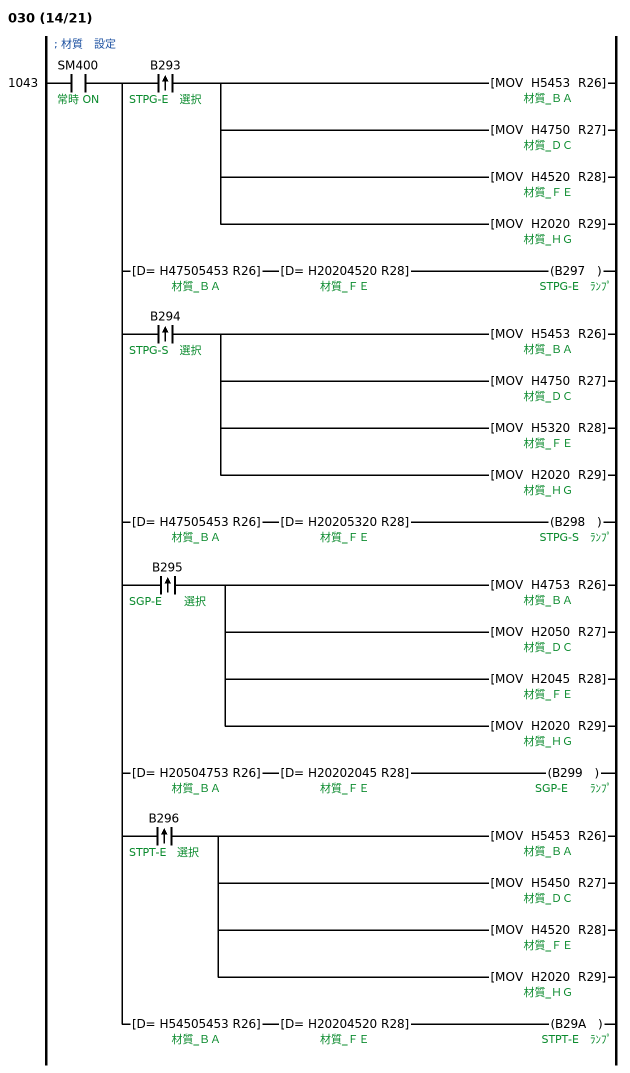
; 材質　設定
1043  LD      SM400  ; 常時 ON
      MPS
      ANDP    B293  ; STPG-E　選択
      MOV     H5453 R26  ; 材質_ＢＡ
      MOV     H4750 R27  ; 材質_ＤＣ
      MOV     H4520 R28  ; 材質_ＦＥ
      MOV     H2020 R29  ; 材質_ＨＧ
      MRD
      ANDD=   H47505453 R26  ; 材質_ＢＡ
      ANDD=   H20204520 R28  ; 材質_ＦＥ
      OUT     B297  ; STPG-E　ﾗﾝﾌﾟ
      MRD
      ANDP    B294  ; STPG-S　選択
      MOV     H5453 R26
      MOV     H4750 R27
      MOV     H5320 R28
      MOV     H2020 R29
      MRD
      ANDD=   H47505453 R26  ; 材質_ＢＡ
      ANDD=   H20205320 R28  ; 材質_ＦＥ
      OUT     B298  ; STPG-S　ﾗﾝﾌﾟ
      MRD
      ANDP    B295  ; SGP-E　　選択
      MOV     H4753 R26
      MOV     H2050 R27
      MOV     H2045 R28
      MOV     H2020 R29
      MRD
      ANDD=   H20504753 R26  ; 材質_ＢＡ
      ANDD=   H20202045 R28  ; 材質_ＦＥ
      OUT     B299  ; SGP-E　　ﾗﾝﾌﾟ
      MRD
      ANDP    B296  ; STPT-E　選択
      MOV     H5453 R26
      MOV     H5450 R27
      MOV     H4520 R28
      MOV     H2020 R29
      MPP
      ANDD=   H54505453 R26  ; 材質_ＢＡ
      ANDD=   H20204520 R28  ; 材質_ＦＥ
      OUT     B29A  ; STPT-E　ﾗﾝﾌﾟ
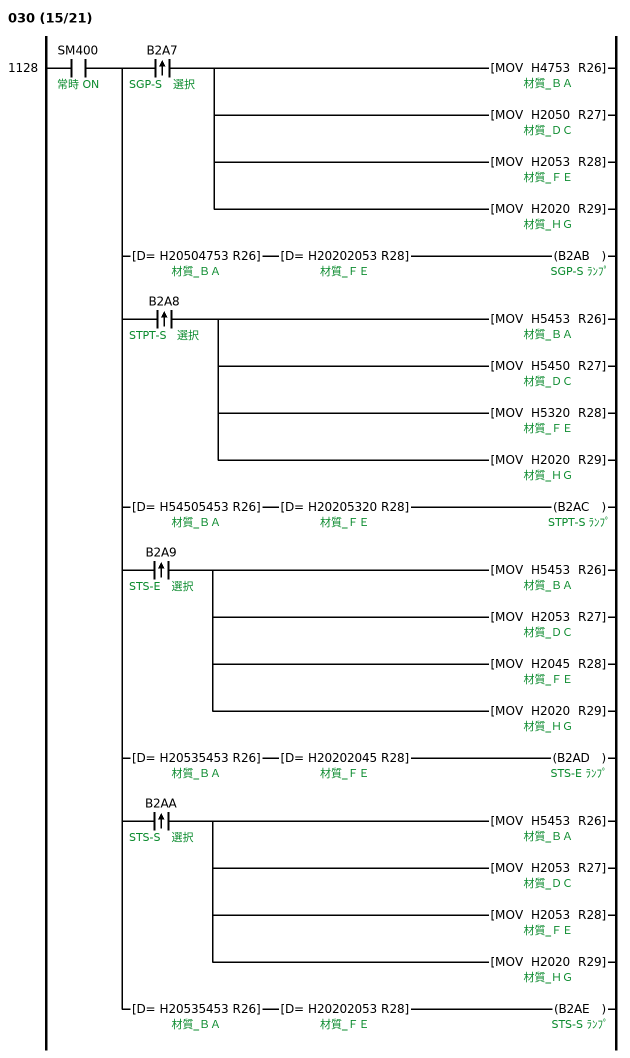
1128  LD      SM400  ; 常時 ON
      MPS
      ANDP    B2A7  ; SGP-S　選択
      MOV     H4753 R26
      MOV     H2050 R27
      MOV     H2053 R28
      MOV     H2020 R29
      MRD
      ANDD=   H20504753 R26  ; 材質_ＢＡ
      ANDD=   H20202053 R28  ; 材質_ＦＥ
      OUT     B2AB  ; SGP-S ﾗﾝﾌﾟ
      MRD
      ANDP    B2A8  ; STPT-S　選択
      MOV     H5453 R26
      MOV     H5450 R27
      MOV     H5320 R28
      MOV     H2020 R29
      MRD
      ANDD=   H54505453 R26  ; 材質_ＢＡ
      ANDD=   H20205320 R28  ; 材質_ＦＥ
      OUT     B2AC  ; STPT-S ﾗﾝﾌﾟ
      MRD
      ANDP    B2A9  ; STS-E　選択
      MOV     H5453 R26
      MOV     H2053 R27
      MOV     H2045 R28
      MOV     H2020 R29
      MRD
      ANDD=   H20535453 R26  ; 材質_ＢＡ
      ANDD=   H20202045 R28  ; 材質_ＦＥ
      OUT     B2AD  ; STS-E ﾗﾝﾌﾟ
      MRD
      ANDP    B2AA  ; STS-S　選択
      MOV     H5453 R26
      MOV     H2053 R27
      MOV     H2053 R28
      MOV     H2020 R29
      MPP
      ANDD=   H20535453 R26  ; 材質_ＢＡ
      ANDD=   H20202053 R28  ; 材質_ＦＥ
      OUT     B2AE  ; STS-S ﾗﾝﾌﾟ
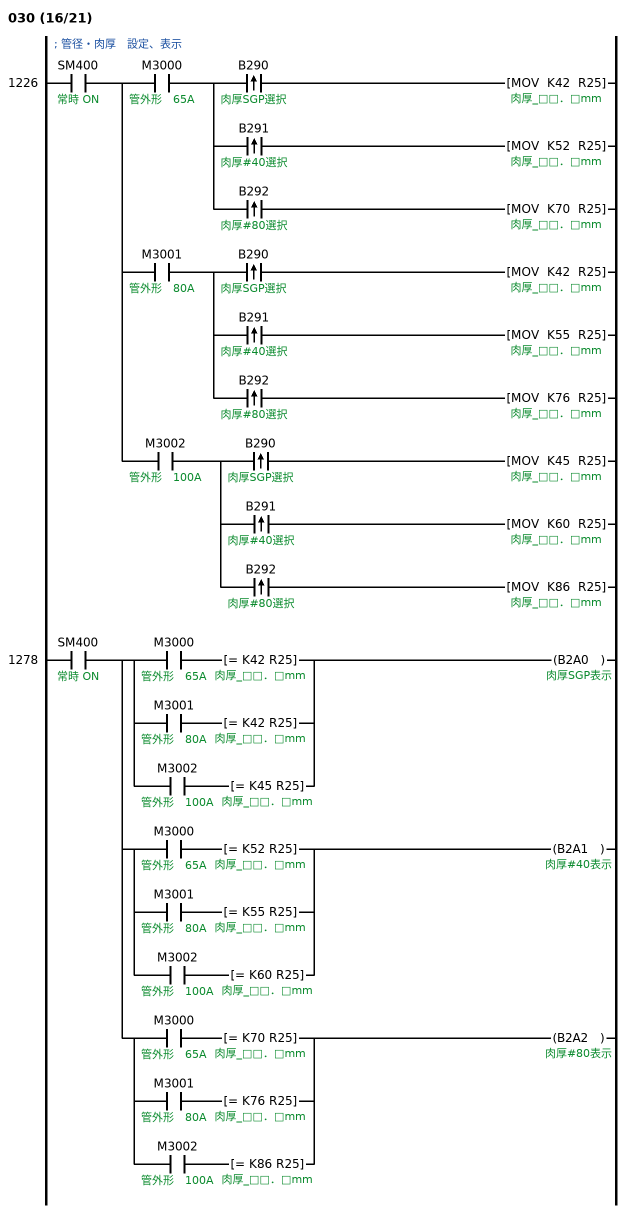
; 管径・肉厚　設定、表示
1226  LD      SM400  ; 常時 ON
      MPS
      AND     M3000  ; 管外形　65A
      MPS
      ANDP    B290  ; 肉厚SGP選択
      MOV     K42 R25  ; 肉厚_□□．□mm
      MRD
      ANDP    B291  ; 肉厚#40選択
      MOV     K52 R25
      MPP
      ANDP    B292  ; 肉厚#80選択
      MOV     K70 R25
      MRD
      AND     M3001  ; 管外形　80A
      MPS
      ANDP    B290  ; 肉厚SGP選択
      MOV     K42 R25
      MRD
      ANDP    B291  ; 肉厚#40選択
      MOV     K55 R25
      MPP
      ANDP    B292  ; 肉厚#80選択
      MOV     K76 R25
      MPP
      AND     M3002  ; 管外形　100A
      MPS
      ANDP    B290  ; 肉厚SGP選択
      MOV     K45 R25
      MRD
      ANDP    B291  ; 肉厚#40選択
      MOV     K60 R25
      MPP
      ANDP    B292  ; 肉厚#80選択
      MOV     K86 R25
1278  LD      SM400  ; 常時 ON
      MPS
      LD      M3000  ; 管外形　65A
      AND=    K42 R25  ; 肉厚_□□．□mm
      LD      M3001  ; 管外形　80A
      AND=    K42 R25  ; 肉厚_□□．□mm
      ORB
      LD      M3002  ; 管外形　100A
      AND=    K45 R25  ; 肉厚_□□．□mm
      ORB
      ANB
      OUT     B2A0  ; 肉厚SGP表示
      MRD
      LD      M3000  ; 管外形　65A
      AND=    K52 R25  ; 肉厚_□□．□mm
      LD      M3001  ; 管外形　80A
      AND=    K55 R25  ; 肉厚_□□．□mm
      ORB
      LD      M3002  ; 管外形　100A
      AND=    K60 R25  ; 肉厚_□□．□mm
      ORB
      ANB
      OUT     B2A1  ; 肉厚#40表示
      MPP
      LD      M3000  ; 管外形　65A
      AND=    K70 R25  ; 肉厚_□□．□mm
      LD      M3001  ; 管外形　80A
      AND=    K76 R25  ; 肉厚_□□．□mm
      ORB
      LD      M3002  ; 管外形　100A
      AND=    K86 R25  ; 肉厚_□□．□mm
      ORB
      ANB
      OUT     B2A2  ; 肉厚#80表示
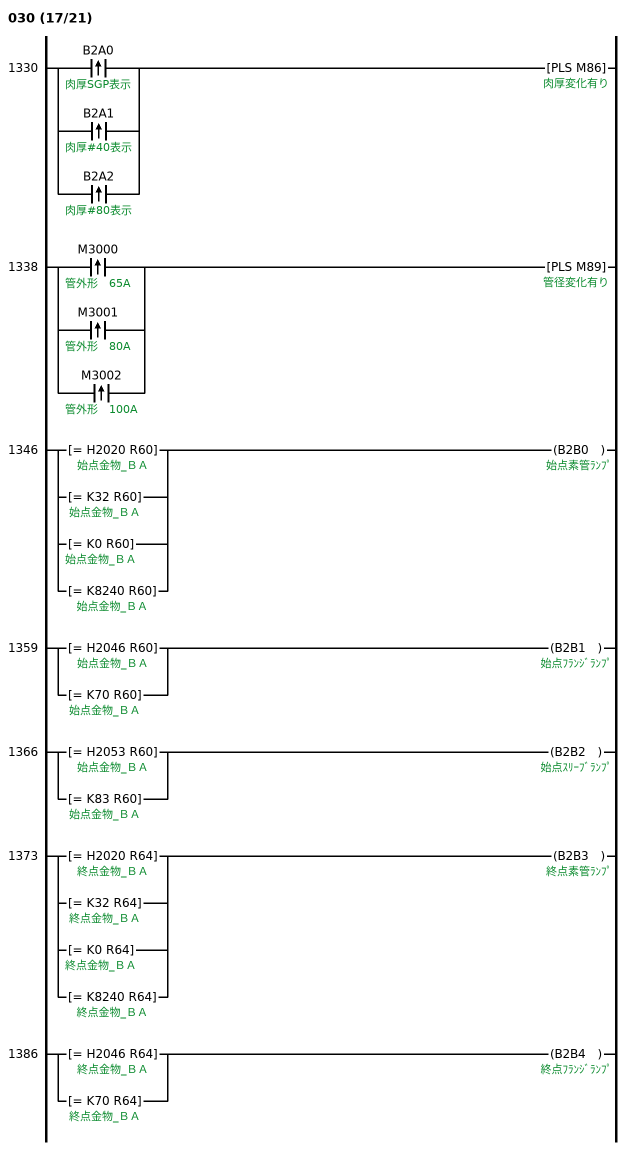
1330  LDP     B2A0  ; 肉厚SGP表示
      ORP     B2A1  ; 肉厚#40表示
      ORP     B2A2  ; 肉厚#80表示
      PLS     M86  ; 肉厚変化有り
1338  LDP     M3000  ; 管外形　65A
      ORP     M3001  ; 管外形　80A
      ORP     M3002  ; 管外形　100A
      PLS     M89  ; 管径変化有り
1346  LD=     H2020 R60  ; 始点金物_ＢＡ
      OR=     K32 R60  ; 始点金物_ＢＡ
      OR=     K0 R60  ; 始点金物_ＢＡ
      OR=     K8240 R60  ; 始点金物_ＢＡ
      OUT     B2B0  ; 始点素管ﾗﾝﾌﾟ
1359  LD=     H2046 R60  ; 始点金物_ＢＡ
      OR=     K70 R60  ; 始点金物_ＢＡ
      OUT     B2B1  ; 始点ﾌﾗﾝｼﾞﾗﾝﾌﾟ
1366  LD=     H2053 R60  ; 始点金物_ＢＡ
      OR=     K83 R60  ; 始点金物_ＢＡ
      OUT     B2B2  ; 始点ｽﾘｰﾌﾞﾗﾝﾌﾟ
1373  LD=     H2020 R64  ; 終点金物_ＢＡ
      OR=     K32 R64  ; 終点金物_ＢＡ
      OR=     K0 R64  ; 終点金物_ＢＡ
      OR=     K8240 R64  ; 終点金物_ＢＡ
      OUT     B2B3  ; 終点素管ﾗﾝﾌﾟ
1386  LD=     H2046 R64  ; 終点金物_ＢＡ
      OR=     K70 R64  ; 終点金物_ＢＡ
      OUT     B2B4  ; 終点ﾌﾗﾝｼﾞﾗﾝﾌﾟ
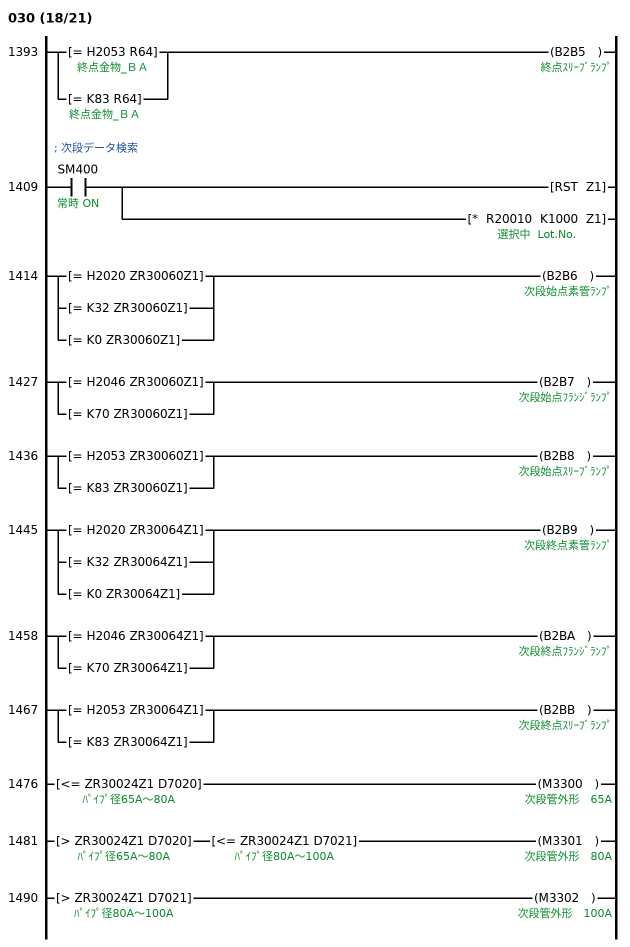
1393  LD=     H2053 R64  ; 終点金物_ＢＡ
      OR=     K83 R64  ; 終点金物_ＢＡ
      OUT     B2B5  ; 終点ｽﾘｰﾌﾞﾗﾝﾌﾟ
; 次段データ検索
1409  LD      SM400  ; 常時 ON
      RST     Z1
      *       R20010 K1000 Z1  ; 選択中  Lot.No.
1414  LD=     H2020 ZR30060Z1
      OR=     K32 ZR30060Z1
      OR=     K0 ZR30060Z1
      OUT     B2B6  ; 次段始点素管ﾗﾝﾌﾟ
1427  LD=     H2046 ZR30060Z1
      OR=     K70 ZR30060Z1
      OUT     B2B7  ; 次段始点ﾌﾗﾝｼﾞﾗﾝﾌﾟ
1436  LD=     H2053 ZR30060Z1
      OR=     K83 ZR30060Z1
      OUT     B2B8  ; 次段始点ｽﾘｰﾌﾞﾗﾝﾌﾟ
1445  LD=     H2020 ZR30064Z1
      OR=     K32 ZR30064Z1
      OR=     K0 ZR30064Z1
      OUT     B2B9  ; 次段終点素管ﾗﾝﾌﾟ
1458  LD=     H2046 ZR30064Z1
      OR=     K70 ZR30064Z1
      OUT     B2BA  ; 次段終点ﾌﾗﾝｼﾞﾗﾝﾌﾟ
1467  LD=     H2053 ZR30064Z1
      OR=     K83 ZR30064Z1
      OUT     B2BB  ; 次段終点ｽﾘｰﾌﾞﾗﾝﾌﾟ
1476  LD<=    ZR30024Z1 D7020  ; ﾊﾟｲﾌﾟ径65A～80A
      OUT     M3300  ; 次段管外形　65A
1481  LD>     ZR30024Z1 D7020  ; ﾊﾟｲﾌﾟ径65A～80A
      AND<=   ZR30024Z1 D7021  ; ﾊﾟｲﾌﾟ径80A～100A
      OUT     M3301  ; 次段管外形　80A
1490  LD>     ZR30024Z1 D7021  ; ﾊﾟｲﾌﾟ径80A～100A
      OUT     M3302  ; 次段管外形　100A
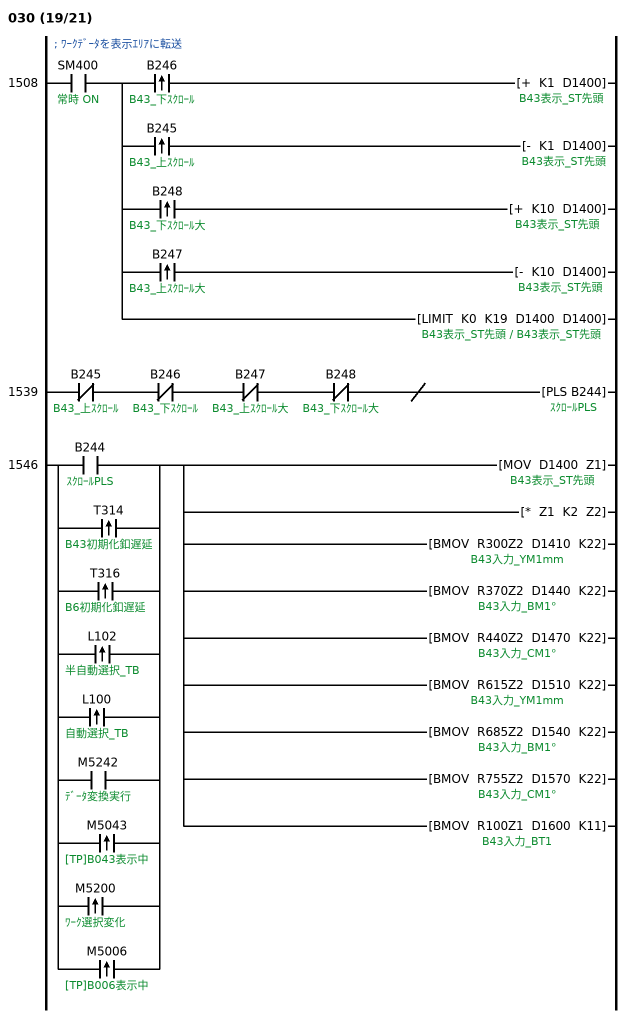
; ﾜｰｸﾃﾞｰﾀを表示ｴﾘｱに転送
1508  LD      SM400  ; 常時 ON
      MPS
      ANDP    B246  ; B43_下ｽｸﾛｰﾙ
      +       K1 D1400  ; B43表示_ST先頭
      MRD
      ANDP    B245  ; B43_上ｽｸﾛｰﾙ
      -       K1 D1400
      MRD
      ANDP    B248  ; B43_下ｽｸﾛｰﾙ大
      +       K10 D1400
      MRD
      ANDP    B247  ; B43_上ｽｸﾛｰﾙ大
      -       K10 D1400
      MPP
      LIMIT   K0 K19 D1400 D1400
1539  LDI     B245  ; B43_上ｽｸﾛｰﾙ
      ANI     B246  ; B43_下ｽｸﾛｰﾙ
      ANI     B247  ; B43_上ｽｸﾛｰﾙ大
      ANI     B248  ; B43_下ｽｸﾛｰﾙ大
      INV
      PLS     B244  ; ｽｸﾛｰﾙPLS
1546  LD      B244  ; ｽｸﾛｰﾙPLS
      ORP     T314  ; B43初期化釦遅延
      ORP     T316  ; B6初期化釦遅延
      ORP     L102  ; 半自動選択_TB
      ORP     L100  ; 自動選択_TB
      OR      M5242  ; ﾃﾞｰﾀ変換実行
      ORP     M5043  ; [TP]B043表示中
      ORP     M5200  ; ﾜｰｸ選択変化
      ORP     M5006  ; [TP]B006表示中
      MOV     D1400 Z1
      *       Z1 K2 Z2
      BMOV    R300Z2 D1410 K22  ; B43入力_YM1mm
      BMOV    R370Z2 D1440 K22  ; B43入力_BM1°
      BMOV    R440Z2 D1470 K22  ; B43入力_CM1°
      BMOV    R615Z2 D1510 K22  ; B43入力_YM1mm
      BMOV    R685Z2 D1540 K22  ; B43入力_BM1°
      BMOV    R755Z2 D1570 K22  ; B43入力_CM1°
      BMOV    R100Z1 D1600 K11  ; B43入力_BT1
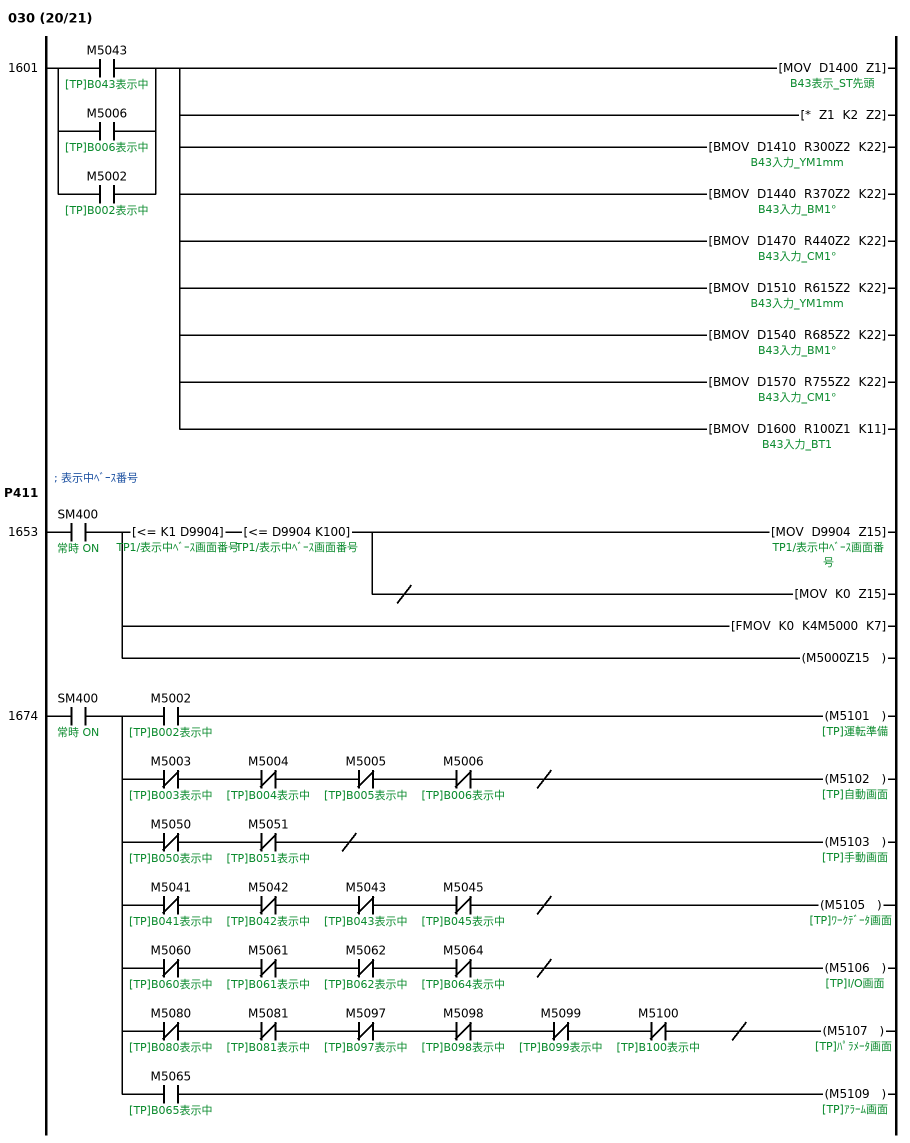
1601  LD      M5043  ; [TP]B043表示中
      OR      M5006  ; [TP]B006表示中
      OR      M5002  ; [TP]B002表示中
      MOV     D1400 Z1
      *       Z1 K2 Z2
      BMOV    D1410 R300Z2 K22
      BMOV    D1440 R370Z2 K22
      BMOV    D1470 R440Z2 K22
      BMOV    D1510 R615Z2 K22
      BMOV    D1540 R685Z2 K22
      BMOV    D1570 R755Z2 K22
      BMOV    D1600 R100Z1 K11
; 表示中ﾍﾞｰｽ番号
      P411
1653  LD      SM400  ; 常時 ON
      MPS
      AND<=   K1 D9904  ; TP1/表示中ﾍﾞｰｽ画面番号
      AND<=   D9904 K100  ; TP1/表示中ﾍﾞｰｽ画面番号
      MOV     D9904 Z15
      INV
      MOV     K0 Z15
      MPP
      FMOV    K0 K4M5000 K7  ; [TP]B00表示先頭
      OUT     M5000Z15
1674  LD      SM400  ; 常時 ON
      MPS
      AND     M5002  ; [TP]B002表示中
      OUT     M5101  ; [TP]運転準備
      MRD
      ANI     M5003  ; [TP]B003表示中
      ANI     M5004  ; [TP]B004表示中
      ANI     M5005  ; [TP]B005表示中
      ANI     M5006  ; [TP]B006表示中
      INV
      OUT     M5102  ; [TP]自動画面
      MRD
      ANI     M5050  ; [TP]B050表示中
      ANI     M5051  ; [TP]B051表示中
      INV
      OUT     M5103  ; [TP]手動画面
      MRD
      ANI     M5041  ; [TP]B041表示中
      ANI     M5042  ; [TP]B042表示中
      ANI     M5043  ; [TP]B043表示中
      ANI     M5045  ; [TP]B045表示中
      INV
      OUT     M5105  ; [TP]ﾜｰｸﾃﾞｰﾀ画面
      MRD
      ANI     M5060  ; [TP]B060表示中
      ANI     M5061  ; [TP]B061表示中
      ANI     M5062  ; [TP]B062表示中
      ANI     M5064  ; [TP]B064表示中
      INV
      OUT     M5106  ; [TP]I/O画面
      MRD
      ANI     M5080  ; [TP]B080表示中
      ANI     M5081  ; [TP]B081表示中
      ANI     M5097  ; [TP]B097表示中
      ANI     M5098  ; [TP]B098表示中
      ANI     M5099  ; [TP]B099表示中
      ANI     M5100  ; [TP]B100表示中
      INV
      OUT     M5107  ; [TP]ﾊﾟﾗﾒｰﾀ画面
      MPP
      AND     M5065  ; [TP]B065表示中
      OUT     M5109  ; [TP]ｱﾗｰﾑ画面
; 表示中ｳｨﾝﾄﾞｳ番号
      P412
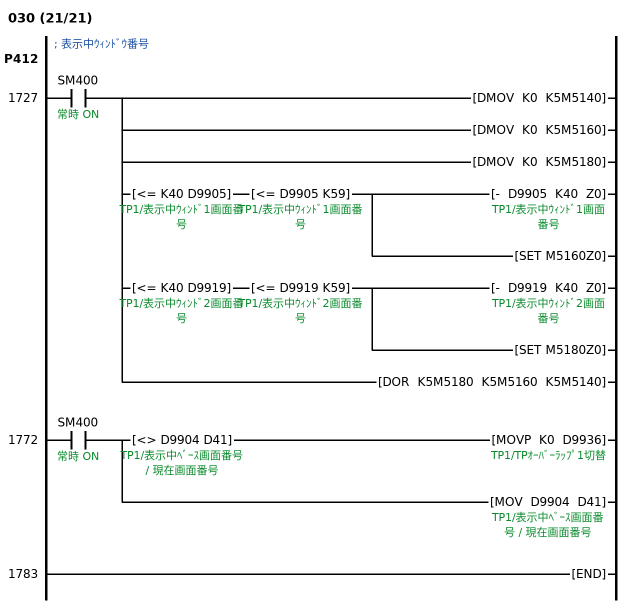
1727  LD      SM400  ; 常時 ON
      DMOV    K0 K5M5140  ; [TP]W40表示中
      DMOV    K0 K5M5160  ; WIN1_W40表示中
      DMOV    K0 K5M5180  ; WIN2_W40表示中
      MPS
      AND<=   K40 D9905  ; TP1/表示中ｳｨﾝﾄﾞ1画面番号
      AND<=   D9905 K59  ; TP1/表示中ｳｨﾝﾄﾞ1画面番号
      -       D9905 K40 Z0
      SET     M5160Z0
      MRD
      AND<=   K40 D9919  ; TP1/表示中ｳｨﾝﾄﾞ2画面番号
      AND<=   D9919 K59  ; TP1/表示中ｳｨﾝﾄﾞ2画面番号
      -       D9919 K40 Z0
      SET     M5180Z0
      MPP
      DOR     K5M5180 K5M5160 K5M5140
1772  LD      SM400  ; 常時 ON
      MPS
      AND<>   D9904 D41  ; TP1/表示中ﾍﾞｰｽ画面番号 / 現在画面番号
      MOVP    K0 D9936
      MPP
      MOV     D9904 D41
1783  END
END_PROGRAM

PROGRAM 031
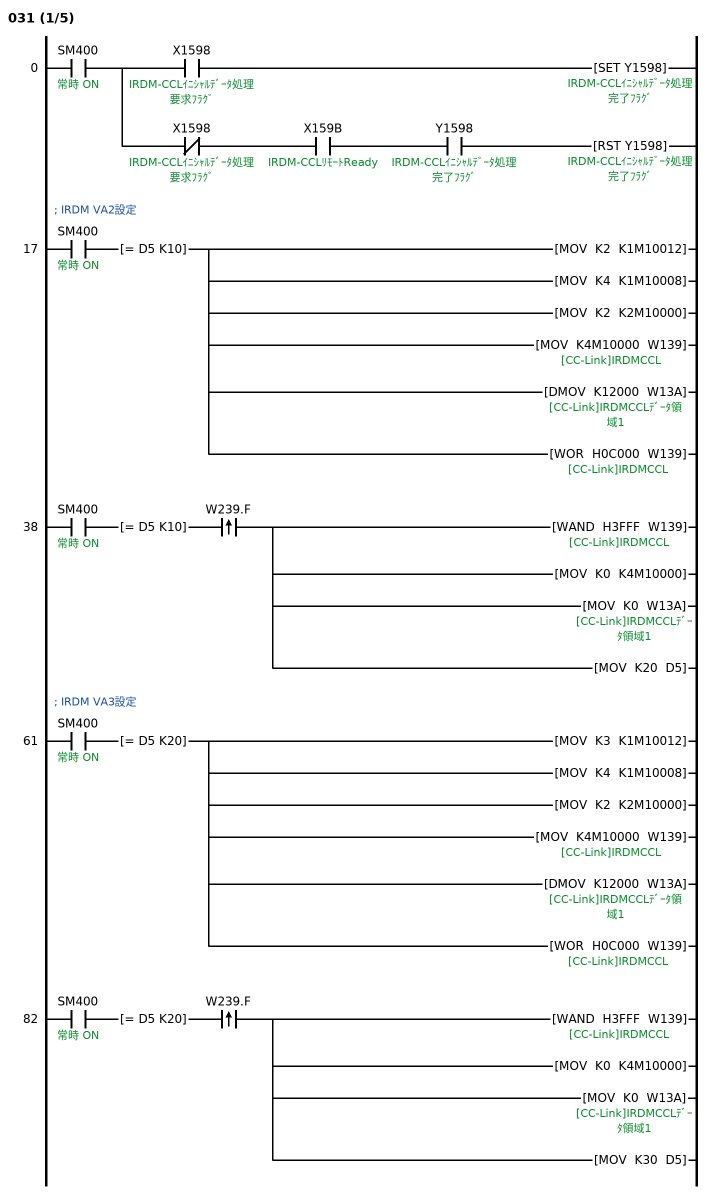
0     LD      SM400  ; 常時 ON
      MPS
      AND     X1598  ; IRDM-CCLｲﾆｼｬﾙﾃﾞｰﾀ処理要求ﾌﾗｸﾞ
      SET     Y1598  ; IRDM-CCLｲﾆｼｬﾙﾃﾞｰﾀ処理完了ﾌﾗｸﾞ
      MPP
      ANI     X1598  ; IRDM-CCLｲﾆｼｬﾙﾃﾞｰﾀ処理要求ﾌﾗｸﾞ
      AND     X159B  ; IRDM-CCLﾘﾓｰﾄReady
      AND     Y1598  ; IRDM-CCLｲﾆｼｬﾙﾃﾞｰﾀ処理完了ﾌﾗｸﾞ
      RST     Y1598  ; IRDM-CCLｲﾆｼｬﾙﾃﾞｰﾀ処理完了ﾌﾗｸﾞ
; IRDM VA2設定
17    LD      SM400  ; 常時 ON
      AND=    D5 K10
      MOV     K2 K1M10012  ; [IRDM仮変数]ﾁｬﾝﾈﾙ番号
      MOV     K4 K1M10008  ; [IRDM仮変数]ｸﾞﾙｰﾌﾟ番号
      MOV     K2 K2M10000  ; [IRDM仮変数]ｲﾝﾃﾞｯｸｽ番号
      MOV     K4M10000 W139  ; [CC-Link]IRDMCCL
      DMOV    K12000 W13A  ; [CC-Link]IRDMCCLﾃﾞｰﾀ領域1
      WOR     H0C000 W139
38    LD      SM400  ; 常時 ON
      AND=    D5 K10
      ANDP    W239.F
      WAND    H3FFF W139
      MOV     K0 K4M10000
      MOV     K0 W13A
      MOV     K20 D5
; IRDM VA3設定
61    LD      SM400  ; 常時 ON
      AND=    D5 K20
      MOV     K3 K1M10012
      MOV     K4 K1M10008
      MOV     K2 K2M10000
      MOV     K4M10000 W139
      DMOV    K12000 W13A
      WOR     H0C000 W139
82    LD      SM400  ; 常時 ON
      AND=    D5 K20
      ANDP    W239.F
      WAND    H3FFF W139
      MOV     K0 K4M10000
      MOV     K0 W13A
      MOV     K30 D5
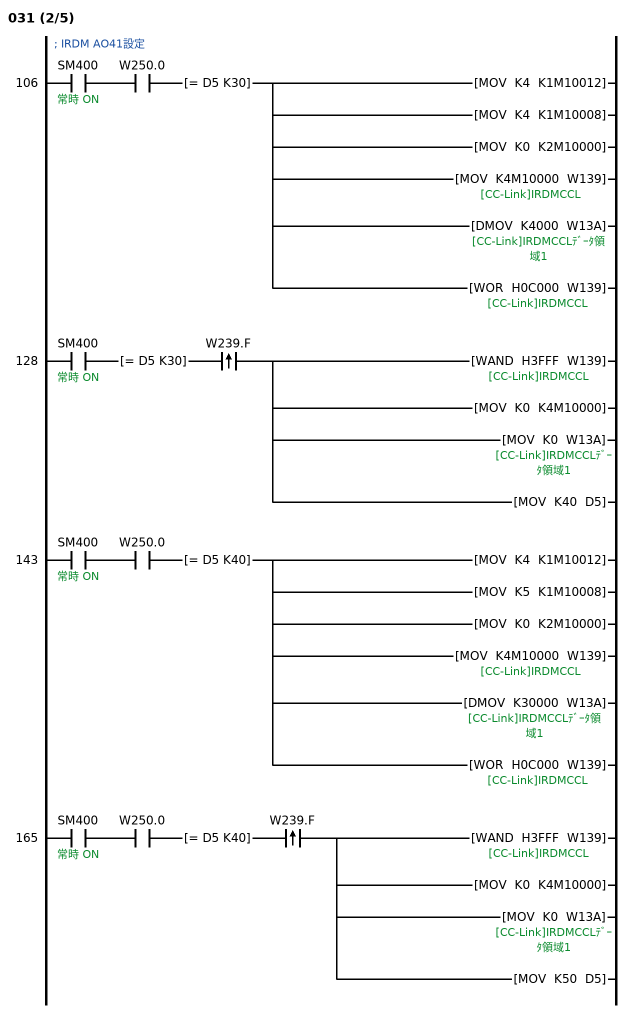
; IRDM AO41設定
106   LD      SM400  ; 常時 ON
      AND     W250.0
      AND=    D5 K30
      MOV     K4 K1M10012
      MOV     K4 K1M10008
      MOV     K0 K2M10000
      MOV     K4M10000 W139
      DMOV    K4000 W13A
      WOR     H0C000 W139
128   LD      SM400  ; 常時 ON
      AND=    D5 K30
      ANDP    W239.F
      WAND    H3FFF W139
      MOV     K0 K4M10000
      MOV     K0 W13A
      MOV     K40 D5
143   LD      SM400  ; 常時 ON
      AND     W250.0
      AND=    D5 K40
      MOV     K4 K1M10012
      MOV     K5 K1M10008
      MOV     K0 K2M10000
      MOV     K4M10000 W139
      DMOV    K30000 W13A
      WOR     H0C000 W139
165   LD      SM400  ; 常時 ON
      AND     W250.0
      AND=    D5 K40
      ANDP    W239.F
      WAND    H3FFF W139
      MOV     K0 K4M10000
      MOV     K0 W13A
      MOV     K50 D5
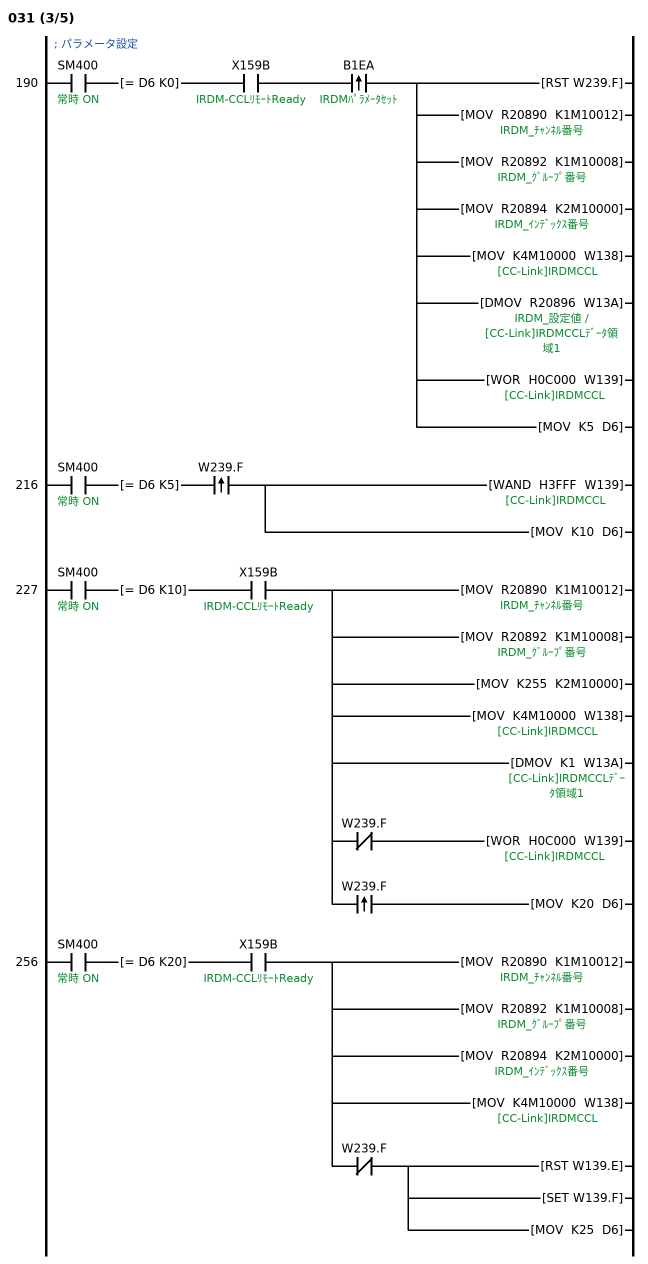
; パラメータ設定
190   LD      SM400  ; 常時 ON
      AND=    D6 K0
      AND     X159B  ; IRDM-CCLﾘﾓｰﾄReady
      ANDP    B1EA  ; IRDMﾊﾟﾗﾒｰﾀｾｯﾄ
      RST     W239.F
      MOV     R20890 K1M10012  ; IRDM_ﾁｬﾝﾈﾙ番号
      MOV     R20892 K1M10008  ; IRDM_ｸﾞﾙｰﾌﾟ番号
      MOV     R20894 K2M10000  ; IRDM_ｲﾝﾃﾞｯｸｽ番号
      MOV     K4M10000 W138  ; [CC-Link]IRDMCCL
      DMOV    R20896 W13A  ; IRDM_設定値
      WOR     H0C000 W139
      MOV     K5 D6
216   LD      SM400  ; 常時 ON
      AND=    D6 K5
      ANDP    W239.F
      WAND    H3FFF W139
      MOV     K10 D6
227   LD      SM400  ; 常時 ON
      AND=    D6 K10
      AND     X159B  ; IRDM-CCLﾘﾓｰﾄReady
      MOV     R20890 K1M10012
      MOV     R20892 K1M10008
      MOV     K255 K2M10000
      MOV     K4M10000 W138
      DMOV    K1 W13A
      MPS
      ANI     W239.F
      WOR     H0C000 W139
      MPP
      ANDP    W239.F
      MOV     K20 D6
256   LD      SM400  ; 常時 ON
      AND=    D6 K20
      AND     X159B  ; IRDM-CCLﾘﾓｰﾄReady
      MOV     R20890 K1M10012
      MOV     R20892 K1M10008
      MOV     R20894 K2M10000
      MOV     K4M10000 W138
      ANI     W239.F
      RST     W139.E
      SET     W139.F
      MOV     K25 D6
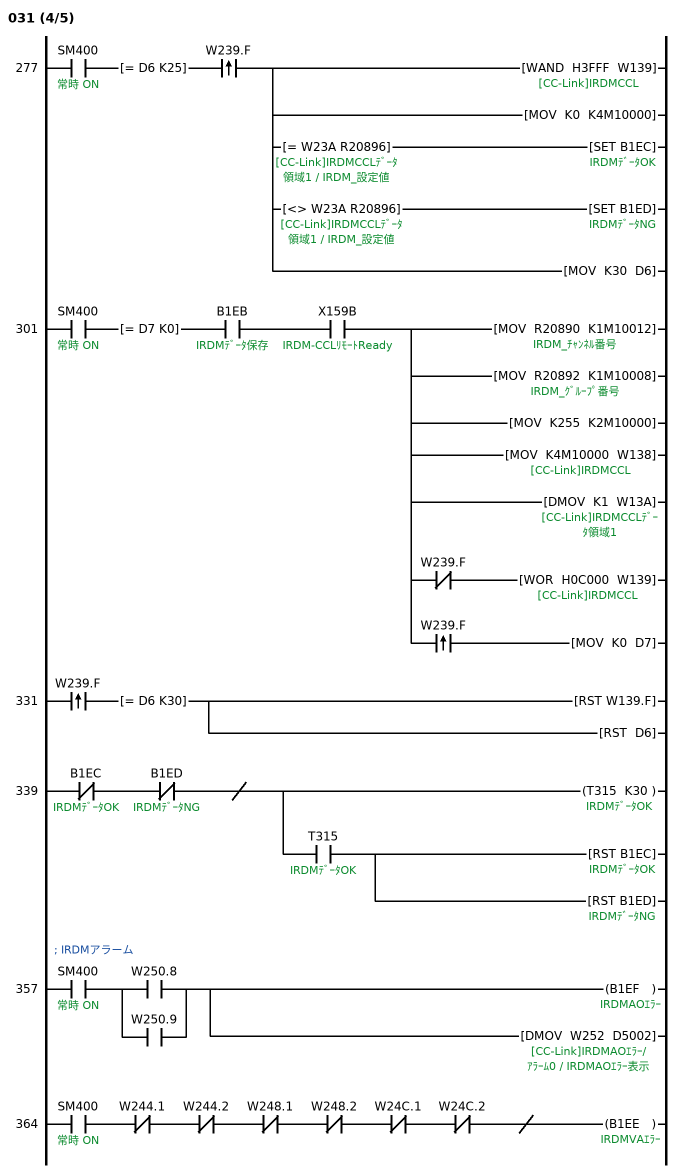
277   LD      SM400  ; 常時 ON
      AND=    D6 K25
      ANDP    W239.F
      WAND    H3FFF W139
      MOV     K0 K4M10000
      MPS
      AND=    W23A R20896  ; [CC-Link]IRDMCCLﾃﾞｰﾀ領域1 / IRDM_設定値
      SET     B1EC  ; IRDMﾃﾞｰﾀOK
      MRD
      AND<>   W23A R20896  ; [CC-Link]IRDMCCLﾃﾞｰﾀ領域1 / IRDM_設定値
      SET     B1ED  ; IRDMﾃﾞｰﾀNG
      MPP
      MOV     K30 D6
301   LD      SM400  ; 常時 ON
      AND=    D7 K0
      AND     B1EB  ; IRDMﾃﾞｰﾀ保存
      AND     X159B  ; IRDM-CCLﾘﾓｰﾄReady
      MOV     R20890 K1M10012
      MOV     R20892 K1M10008
      MOV     K255 K2M10000
      MOV     K4M10000 W138
      DMOV    K1 W13A
      MPS
      ANI     W239.F
      WOR     H0C000 W139
      MPP
      ANDP    W239.F
      MOV     K0 D7
331   LDP     W239.F
      AND=    D6 K30
      RST     W139.F
      RST     D6
339   LDI     B1EC  ; IRDMﾃﾞｰﾀOK
      ANI     B1ED  ; IRDMﾃﾞｰﾀNG
      INV
      OUT     T315 K30  ; IRDMﾃﾞｰﾀOK
      AND     T315  ; IRDMﾃﾞｰﾀOK
      RST     B1EC  ; IRDMﾃﾞｰﾀOK
      RST     B1ED  ; IRDMﾃﾞｰﾀNG
; IRDMアラーム
357   LD      SM400  ; 常時 ON
      LD      W250.8
      OR      W250.9
      ANB
      OUT     B1EF  ; IRDMAOｴﾗｰ
      DMOV    W252 D5002  ; [CC-Link]IRDMAOｴﾗｰ/ｱﾗｰﾑ0 / IRDMAOｴﾗｰ表示
364   LD      SM400  ; 常時 ON
      ANI     W244.1
      ANI     W244.2
      ANI     W248.1
      ANI     W248.2
      ANI     W24C.1
      ANI     W24C.2
      INV
      OUT     B1EE  ; IRDMVAｴﾗｰ
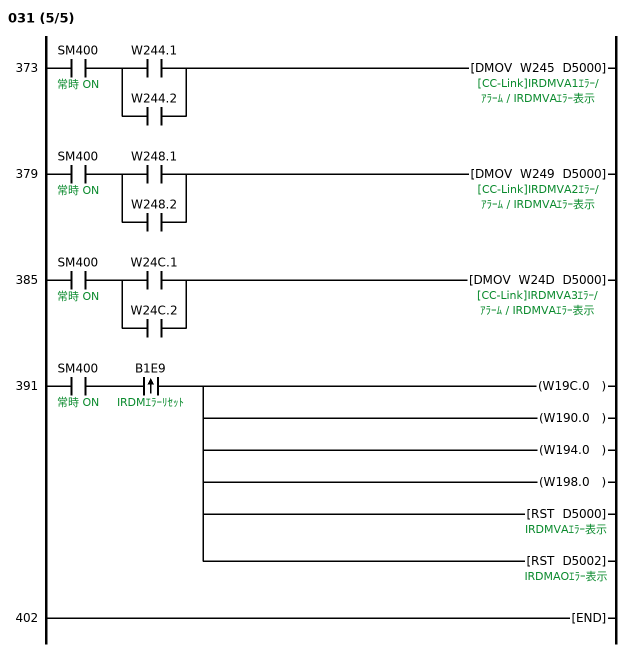
373   LD      SM400  ; 常時 ON
      LD      W244.1
      OR      W244.2
      ANB
      DMOV    W245 D5000  ; [CC-Link]IRDMVA1ｴﾗｰ/ｱﾗｰﾑ / IRDMVAｴﾗｰ表示
379   LD      SM400  ; 常時 ON
      LD      W248.1
      OR      W248.2
      ANB
      DMOV    W249 D5000  ; [CC-Link]IRDMVA2ｴﾗｰ/ｱﾗｰﾑ
385   LD      SM400  ; 常時 ON
      LD      W24C.1
      OR      W24C.2
      ANB
      DMOV    W24D D5000  ; [CC-Link]IRDMVA3ｴﾗｰ/ｱﾗｰﾑ
391   LD      SM400  ; 常時 ON
      ANDP    B1E9  ; IRDMｴﾗｰﾘｾｯﾄ
      OUT     W19C.0
      OUT     W190.0
      OUT     W194.0
      OUT     W198.0
      RST     D5000  ; IRDMVAｴﾗｰ表示
      RST     D5002  ; IRDMAOｴﾗｰ表示
402   END
END_PROGRAM

PROGRAM 016
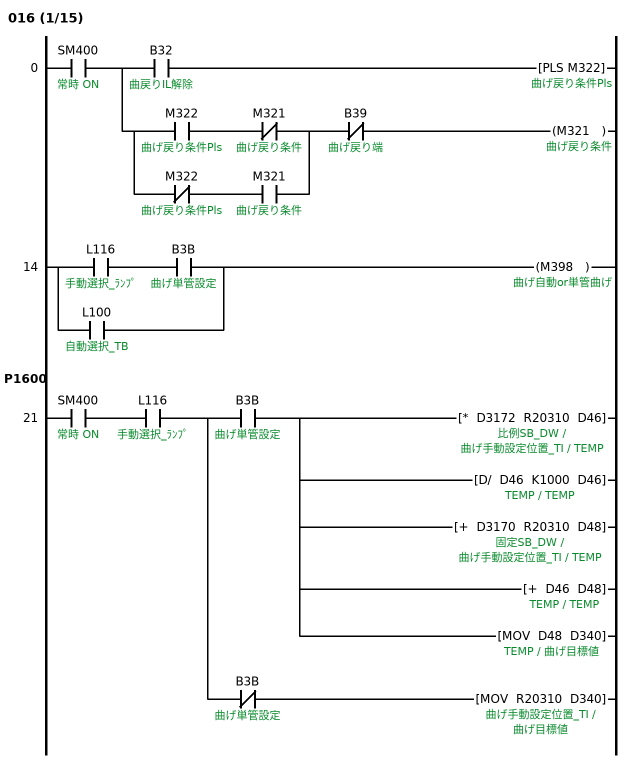
0     LD      SM400  ; 常時 ON
      MPS
      AND     B32  ; 曲戻りIL解除
      PLS     M322  ; 曲げ戻り条件Pls
      MPP
      LD      M322  ; 曲げ戻り条件Pls
      ANI     M321  ; 曲げ戻り条件
      LDI     M322  ; 曲げ戻り条件Pls
      AND     M321  ; 曲げ戻り条件
      ORB
      ANB
      ANI     B39  ; 曲げ戻り端
      OUT     M321  ; 曲げ戻り条件
14    LD      L116  ; 手動選択_ﾗﾝﾌﾟ
      AND     B3B  ; 曲げ単管設定
      OR      L100  ; 自動選択_TB
      OUT     M398  ; 曲げ自動or単管曲げ
; 
      P1600
21    LD      SM400  ; 常時 ON
      AND     L116  ; 手動選択_ﾗﾝﾌﾟ
      MPS
      AND     B3B  ; 曲げ単管設定
      *       D3172 R20310 D46  ; 比例SB_DW / 曲げ手動設定位置_TI / TEMP
      D/      D46 K1000 D46
      +       D3170 R20310 D48  ; 固定SB_DW / TEMP
      +       D46 D48
      MOV     D48 D340  ; 曲げ目標値
      MPP
      ANI     B3B  ; 曲げ単管設定
      MOV     R20310 D340
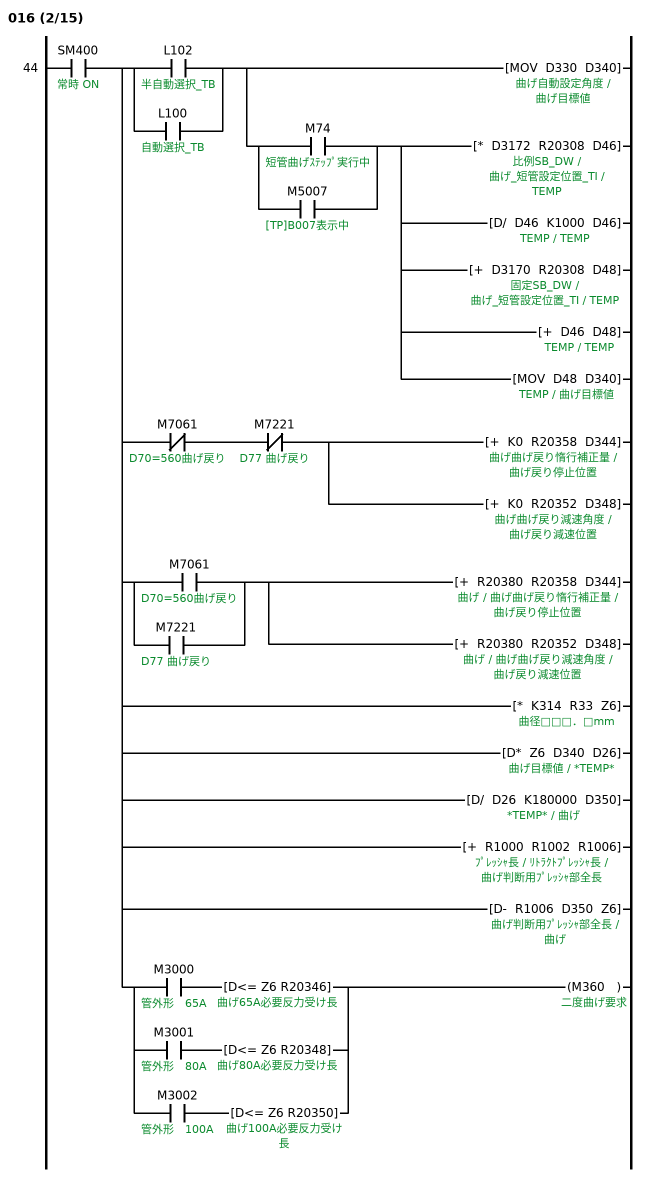
44    LD      SM400  ; 常時 ON
      MPS
      LD      L102  ; 半自動選択_TB
      OR      L100  ; 自動選択_TB
      ANB
      MOV     D330 D340  ; 曲げ自動設定角度
      LD      M74  ; 短管曲げｽﾃｯﾌﾟ実行中
      OR      M5007  ; [TP]B007表示中
      ANB
      *       D3172 R20308 D46  ; 曲げ_短管設定位置_TI
      D/      D46 K1000 D46
      +       D3170 R20308 D48
      +       D46 D48
      MOV     D48 D340
      MRD
      ANI     M7061  ; D70=560曲げ戻り
      ANI     M7221  ; D77 曲げ戻り
      +       K0 R20358 D344  ; 曲げ曲げ戻り惰行補正量 / 曲げ戻り停止位置
      +       K0 R20352 D348  ; 曲げ曲げ戻り減速角度 / 曲げ戻り減速位置
      MRD
      LD      M7061  ; D70=560曲げ戻り
      OR      M7221  ; D77 曲げ戻り
      ANB
      +       R20380 R20358 D344  ; 曲げ
      +       R20380 R20352 D348
      MPP
      *       K314 R33 Z6  ; 曲径□□□．□mm
      D*      Z6 D340 D26  ; *TEMP*
      D/      D26 K180000 D350  ; 曲げ
      +       R1000 R1002 R1006  ; ﾌﾟﾚｯｼｬ長 / ﾘﾄﾗｸﾄﾌﾟﾚｯｼｬ長 / 曲げ判断用ﾌﾟﾚｯｼｬ部全長
      D-      R1006 D350 Z6
      LD      M3000  ; 管外形　65A
      ANDD<=  Z6 R20346  ; 曲げ65A必要反力受け長
      LD      M3001  ; 管外形　80A
      ANDD<=  Z6 R20348  ; 曲げ80A必要反力受け長
      ORB
      LD      M3002  ; 管外形　100A
      ANDD<=  Z6 R20350  ; 曲げ100A必要反力受け長
      ORB
      ANB
      OUT     M360  ; 二度曲げ要求
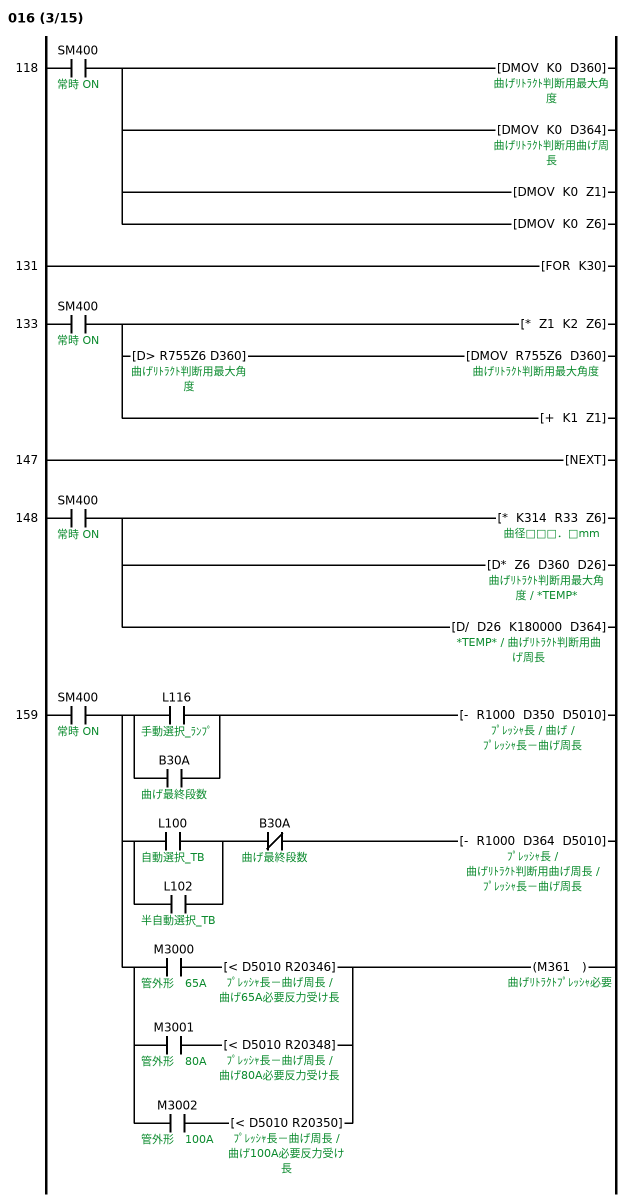
118   LD      SM400  ; 常時 ON
      DMOV    K0 D360  ; 曲げﾘﾄﾗｸﾄ判断用最大角度
      DMOV    K0 D364  ; 曲げﾘﾄﾗｸﾄ判断用曲げ周長
      DMOV    K0 Z1
      DMOV    K0 Z6
131   FOR     K30
133   LD      SM400  ; 常時 ON
      *       Z1 K2 Z6
      MPS
      ANDD>   R755Z6 D360  ; 曲げﾘﾄﾗｸﾄ判断用最大角度
      DMOV    R755Z6 D360
      MPP
      +       K1 Z1
147   NEXT
148   LD      SM400  ; 常時 ON
      *       K314 R33 Z6
      D*      Z6 D360 D26
      D/      D26 K180000 D364
159   LD      SM400  ; 常時 ON
      MPS
      LD      L116  ; 手動選択_ﾗﾝﾌﾟ
      OR      B30A  ; 曲げ最終段数
      ANB
      -       R1000 D350 D5010  ; ﾌﾟﾚｯｼｬ長－曲げ周長
      MRD
      LD      L100  ; 自動選択_TB
      OR      L102  ; 半自動選択_TB
      ANB
      ANI     B30A  ; 曲げ最終段数
      -       R1000 D364 D5010
      MPP
      LD      M3000  ; 管外形　65A
      AND<    D5010 R20346  ; ﾌﾟﾚｯｼｬ長－曲げ周長 / 曲げ65A必要反力受け長
      LD      M3001  ; 管外形　80A
      AND<    D5010 R20348  ; ﾌﾟﾚｯｼｬ長－曲げ周長 / 曲げ80A必要反力受け長
      ORB
      LD      M3002  ; 管外形　100A
      AND<    D5010 R20350  ; ﾌﾟﾚｯｼｬ長－曲げ周長 / 曲げ100A必要反力受け長
      ORB
      ANB
      OUT     M361  ; 曲げﾘﾄﾗｸﾄﾌﾟﾚｯｼｬ必要
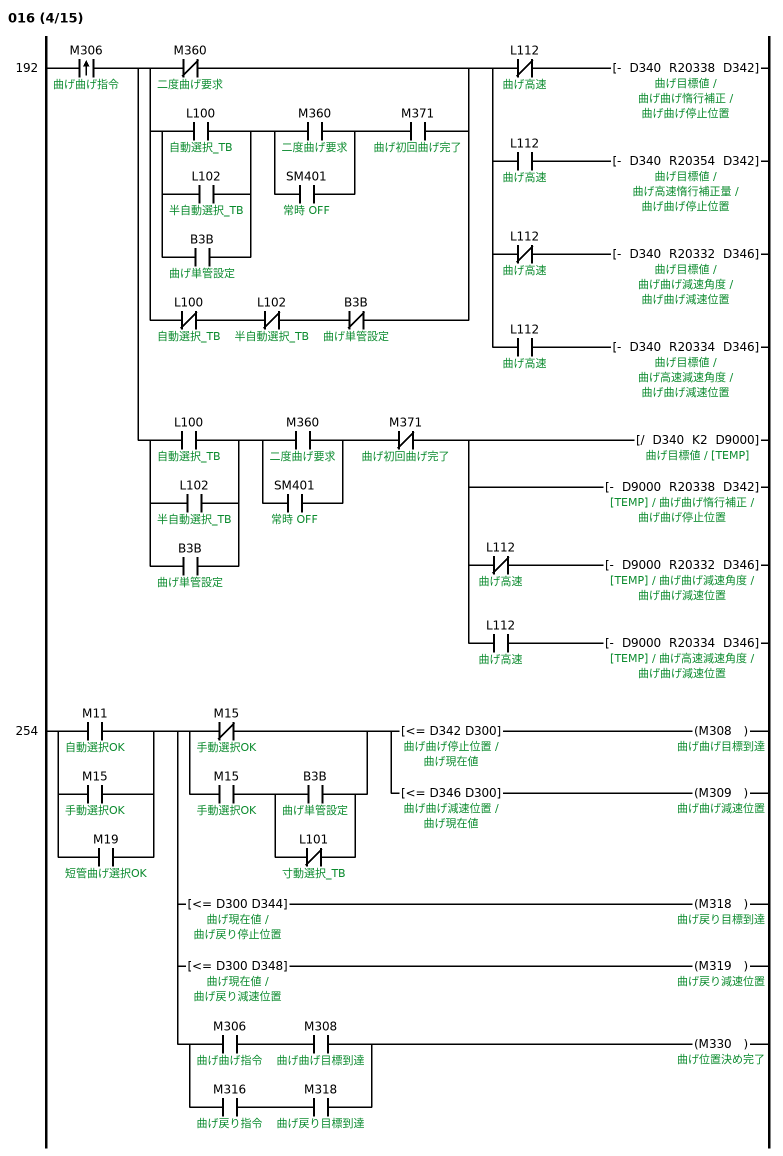
192   LDP     M306  ; 曲げ曲げ指令
      MPS
      LDI     M360  ; 二度曲げ要求
      LD      L100  ; 自動選択_TB
      OR      L102  ; 半自動選択_TB
      OR      B3B  ; 曲げ単管設定
      LD      M360  ; 二度曲げ要求
      OR      SM401  ; 常時 OFF
      ANB
      AND     M371  ; 曲げ初回曲げ完了
      ORB
      LDI     L100  ; 自動選択_TB
      ANI     L102  ; 半自動選択_TB
      ANI     B3B  ; 曲げ単管設定
      ORB
      ANB
      MPS
      ANI     L112  ; 曲げ高速
      -       D340 R20338 D342  ; 曲げ曲げ惰行補正 / 曲げ曲げ停止位置
      MRD
      AND     L112  ; 曲げ高速
      -       D340 R20354 D342  ; 曲げ高速惰行補正量
      MRD
      ANI     L112  ; 曲げ高速
      -       D340 R20332 D346  ; 曲げ曲げ減速角度 / 曲げ曲げ減速位置
      MPP
      AND     L112  ; 曲げ高速
      -       D340 R20334 D346  ; 曲げ高速減速角度
      MPP
      LD      L100  ; 自動選択_TB
      OR      L102  ; 半自動選択_TB
      OR      B3B  ; 曲げ単管設定
      ANB
      LD      M360  ; 二度曲げ要求
      OR      SM401  ; 常時 OFF
      ANB
      ANI     M371  ; 曲げ初回曲げ完了
      /       D340 K2 D9000  ; [TEMP]
      -       D9000 R20338 D342
      MPS
      ANI     L112  ; 曲げ高速
      -       D9000 R20332 D346
      MPP
      AND     L112  ; 曲げ高速
      -       D9000 R20334 D346
254   LD      M11  ; 自動選択OK
      OR      M15  ; 手動選択OK
      OR      M19  ; 短管曲げ選択OK
      MPS
      LDI     M15  ; 手動選択OK
      LD      M15  ; 手動選択OK
      LD      B3B  ; 曲げ単管設定
      ORI     L101  ; 寸動選択_TB
      ANB
      ORB
      ANB
      MPS
      AND<=   D342 D300  ; 曲げ曲げ停止位置 / 曲げ現在値
      OUT     M308  ; 曲げ曲げ目標到達
      MPP
      AND<=   D346 D300  ; 曲げ曲げ減速位置 / 曲げ現在値
      OUT     M309  ; 曲げ曲げ減速位置
      MRD
      AND<=   D300 D344  ; 曲げ現在値 / 曲げ戻り停止位置
      OUT     M318  ; 曲げ戻り目標到達
      MRD
      AND<=   D300 D348  ; 曲げ現在値 / 曲げ戻り減速位置
      OUT     M319  ; 曲げ戻り減速位置
      MPP
      LD      M306  ; 曲げ曲げ指令
      AND     M308  ; 曲げ曲げ目標到達
      LD      M316  ; 曲げ戻り指令
      AND     M318  ; 曲げ戻り目標到達
      ORB
      ANB
      OUT     M330  ; 曲げ位置決め完了
; 
      P1602
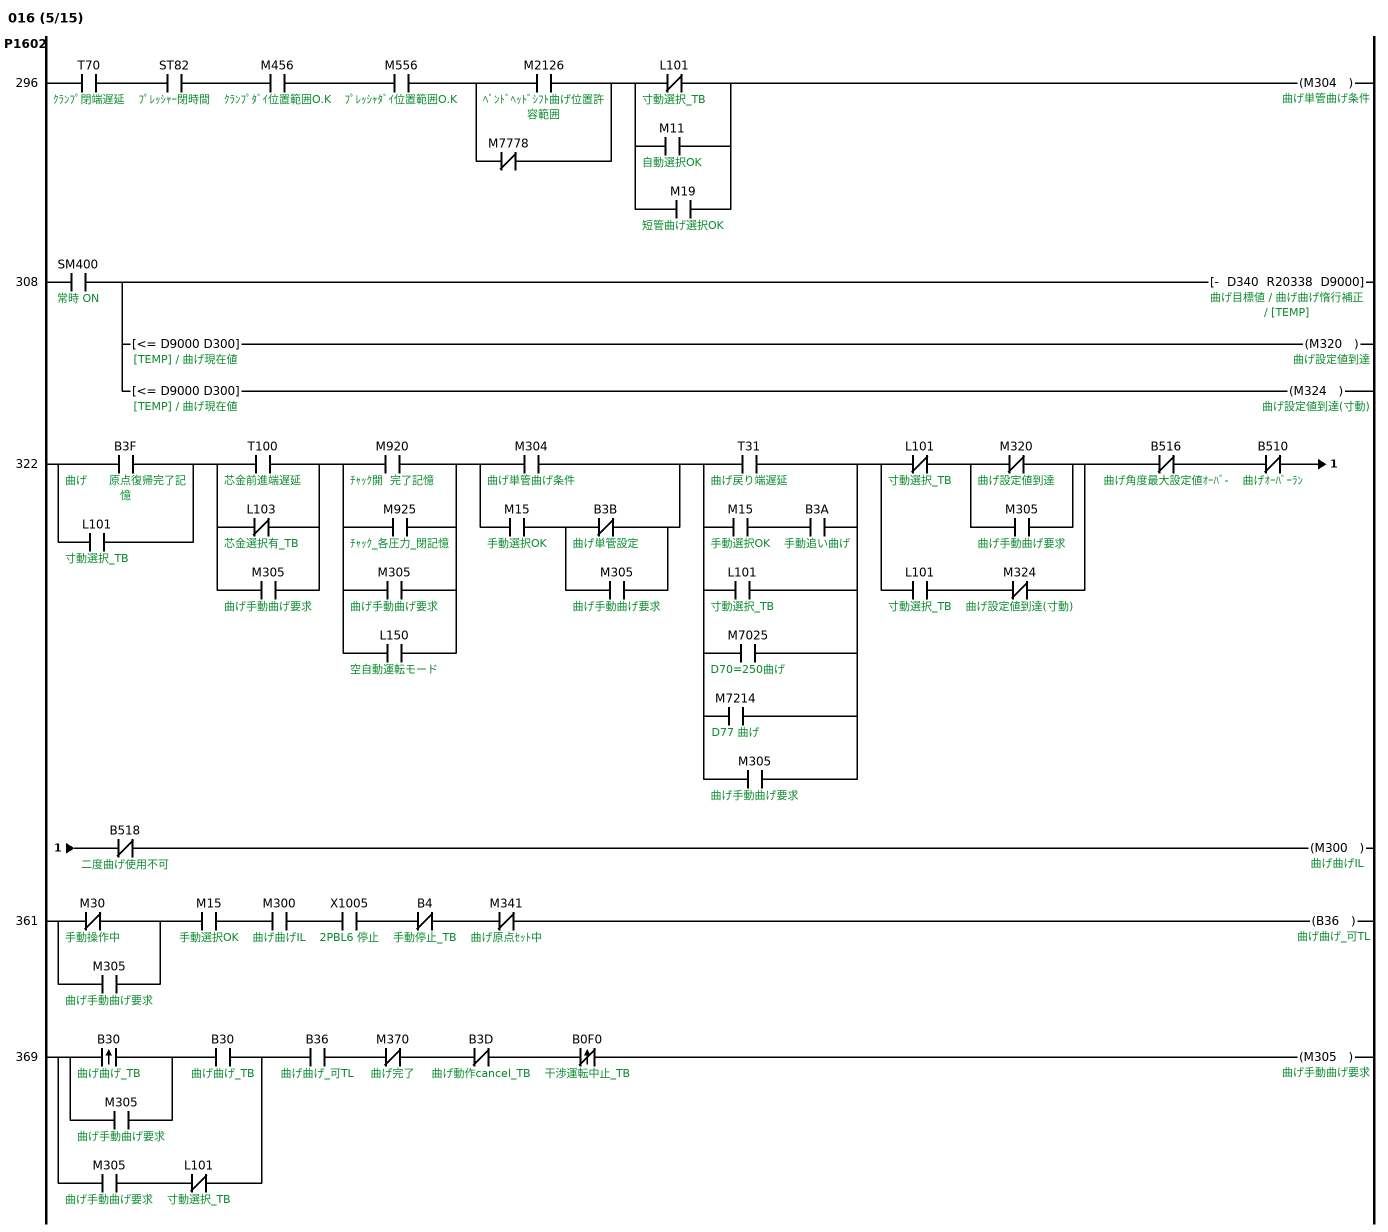
296   LD      T70  ; ｸﾗﾝﾌﾟ閉端遅延
      AND     ST82  ; ﾌﾟﾚｯｼｬｰ閉時間
      AND     M456  ; ｸﾗﾝﾌﾟﾀﾞｲ位置範囲O.K
      AND     M556  ; ﾌﾟﾚｯｼｬﾀﾞｲ位置範囲O.K
      LD      M2126  ; ﾍﾞﾝﾄﾞﾍｯﾄﾞｼﾌﾄ曲げ位置許容範囲
      ORI     M7778
      ANB
      LDI     L101  ; 寸動選択_TB
      OR      M11  ; 自動選択OK
      OR      M19  ; 短管曲げ選択OK
      ANB
      OUT     M304  ; 曲げ単管曲げ条件
308   LD      SM400  ; 常時 ON
      -       D340 R20338 D9000
      MPS
      AND<=   D9000 D300  ; [TEMP] / 曲げ現在値
      OUT     M320  ; 曲げ設定値到達
      MPP
      AND<=   D9000 D300  ; [TEMP] / 曲げ現在値
      OUT     M324  ; 曲げ設定値到達(寸動)
322   LD      B3F  ; 曲げ　　原点復帰完了記憶
      OR      L101  ; 寸動選択_TB
      LD      T100  ; 芯金前進端遅延
      ORI     L103  ; 芯金選択有_TB
      OR      M305  ; 曲げ手動曲げ要求
      ANB
      LD      M920  ; ﾁｬｯｸ開  完了記憶
      OR      M925  ; ﾁｬｯｸ_各圧力_閉記憶
      OR      M305  ; 曲げ手動曲げ要求
      OR      L150  ; 空自動運転モード
      ANB
      LD      M304  ; 曲げ単管曲げ条件
      LD      M15  ; 手動選択OK
      LDI     B3B  ; 曲げ単管設定
      OR      M305  ; 曲げ手動曲げ要求
      ANB
      ORB
      ANB
      LD      T31  ; 曲げ戻り端遅延
      LD      M15  ; 手動選択OK
      AND     B3A  ; 手動追い曲げ
      ORB
      OR      L101  ; 寸動選択_TB
      OR      M7025  ; D70=250曲げ
      OR      M7214  ; D77 曲げ
      OR      M305  ; 曲げ手動曲げ要求
      ANB
      LDI     L101  ; 寸動選択_TB
      LDI     M320  ; 曲げ設定値到達
      OR      M305  ; 曲げ手動曲げ要求
      ANB
      LD      L101  ; 寸動選択_TB
      ANI     M324  ; 曲げ設定値到達(寸動)
      ORB
      ANB
      ANI     B516  ; 曲げ角度最大設定値ｵｰﾊﾞ-
      ANI     B510  ; 曲げｵｰﾊﾞｰﾗﾝ
      ANI     B518  ; 二度曲げ使用不可
      OUT     M300  ; 曲げ曲げIL
361   LDI     M30  ; 手動操作中
      OR      M305  ; 曲げ手動曲げ要求
      AND     M15  ; 手動選択OK
      AND     M300  ; 曲げ曲げIL
      AND     X1005  ; 2PBL6 停止
      ANI     B4  ; 手動停止_TB
      ANI     M341  ; 曲げ原点ｾｯﾄ中
      OUT     B36  ; 曲げ曲げ_可TL
369   LDP     B30  ; 曲げ曲げ_TB
      OR      M305  ; 曲げ手動曲げ要求
      AND     B30  ; 曲げ曲げ_TB
      LD      M305  ; 曲げ手動曲げ要求
      ANI     L101  ; 寸動選択_TB
      ORB
      AND     B36  ; 曲げ曲げ_可TL
      ANI     M370  ; 曲げ完了
      ANI     B3D  ; 曲げ動作cancel_TB
      ANDPI   B0F0  ; 干渉運転中止_TB
      OUT     M305  ; 曲げ手動曲げ要求
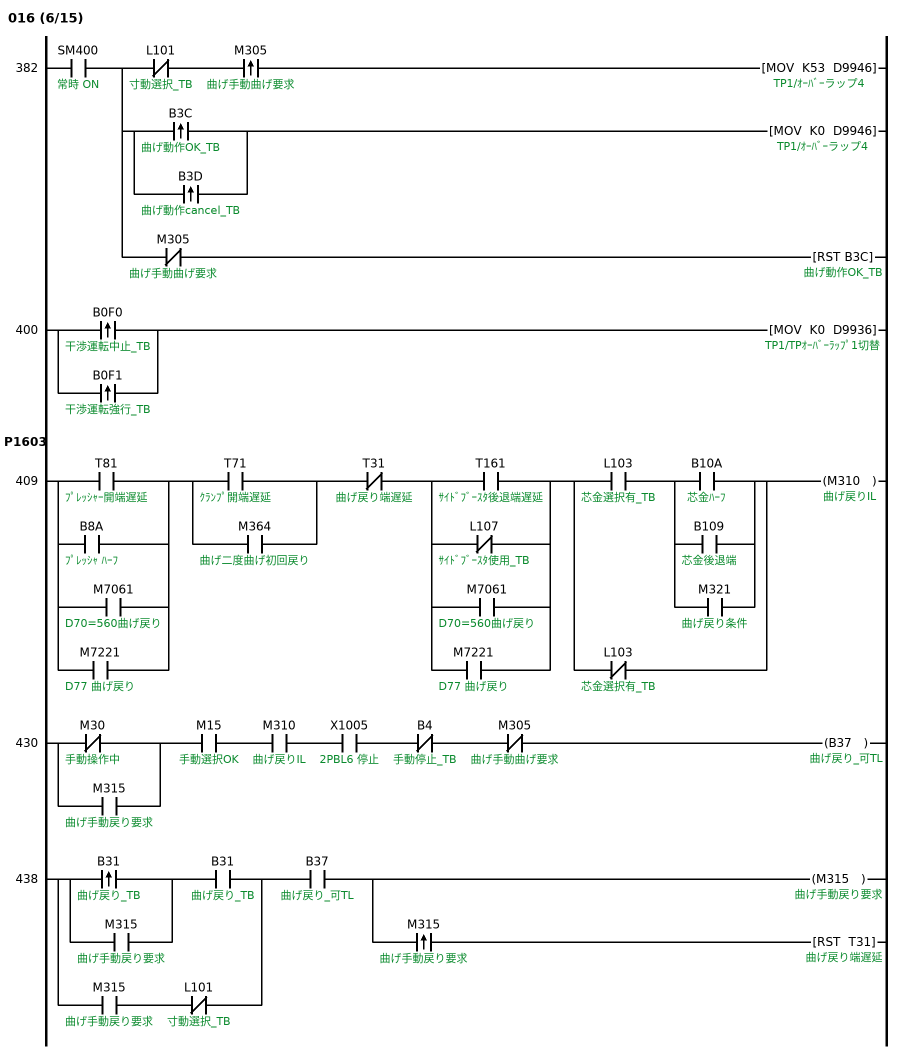
382   LD      SM400  ; 常時 ON
      MPS
      ANI     L101  ; 寸動選択_TB
      ANDP    M305  ; 曲げ手動曲げ要求
      MOV     K53 D9946  ; TP1/ｵｰﾊﾞｰラップ4
      MRD
      LDP     B3C  ; 曲げ動作OK_TB
      ORP     B3D  ; 曲げ動作cancel_TB
      ANB
      MOV     K0 D9946
      MPP
      ANI     M305  ; 曲げ手動曲げ要求
      RST     B3C  ; 曲げ動作OK_TB
400   LDP     B0F0  ; 干渉運転中止_TB
      ORP     B0F1  ; 干渉運転強行_TB
      MOV     K0 D9936  ; TP1/TPｵｰﾊﾞｰﾗｯﾌﾟ1切替
; 
      P1603
409   LD      T81  ; ﾌﾟﾚｯｼｬｰ開端遅延
      OR      B8A  ; ﾌﾟﾚｯｼｬ ﾊｰﾌ
      OR      M7061  ; D70=560曲げ戻り
      OR      M7221  ; D77 曲げ戻り
      LD      T71  ; ｸﾗﾝﾌﾟ開端遅延
      OR      M364  ; 曲げ二度曲げ初回戻り
      ANB
      ANI     T31  ; 曲げ戻り端遅延
      LD      T161  ; ｻｲﾄﾞﾌﾞｰｽﾀ後退端遅延
      ORI     L107  ; ｻｲﾄﾞﾌﾞｰｽﾀ使用_TB
      OR      M7061  ; D70=560曲げ戻り
      OR      M7221  ; D77 曲げ戻り
      ANB
      LD      L103  ; 芯金選択有_TB
      LD      B10A  ; 芯金ﾊｰﾌ
      OR      B109  ; 芯金後退端
      OR      M321  ; 曲げ戻り条件
      ANB
      ORI     L103  ; 芯金選択有_TB
      ANB
      OUT     M310  ; 曲げ戻りIL
430   LDI     M30  ; 手動操作中
      OR      M315  ; 曲げ手動戻り要求
      AND     M15  ; 手動選択OK
      AND     M310  ; 曲げ戻りIL
      AND     X1005  ; 2PBL6 停止
      ANI     B4  ; 手動停止_TB
      ANI     M305  ; 曲げ手動曲げ要求
      OUT     B37  ; 曲げ戻り_可TL
438   LDP     B31  ; 曲げ戻り_TB
      OR      M315  ; 曲げ手動戻り要求
      AND     B31  ; 曲げ戻り_TB
      LD      M315  ; 曲げ手動戻り要求
      ANI     L101  ; 寸動選択_TB
      ORB
      AND     B37  ; 曲げ戻り_可TL
      OUT     M315  ; 曲げ手動戻り要求
      ANDP    M315  ; 曲げ手動戻り要求
      RST     T31  ; 曲げ戻り端遅延
; 曲げｽﾃｯﾌﾟ*********
      P1604
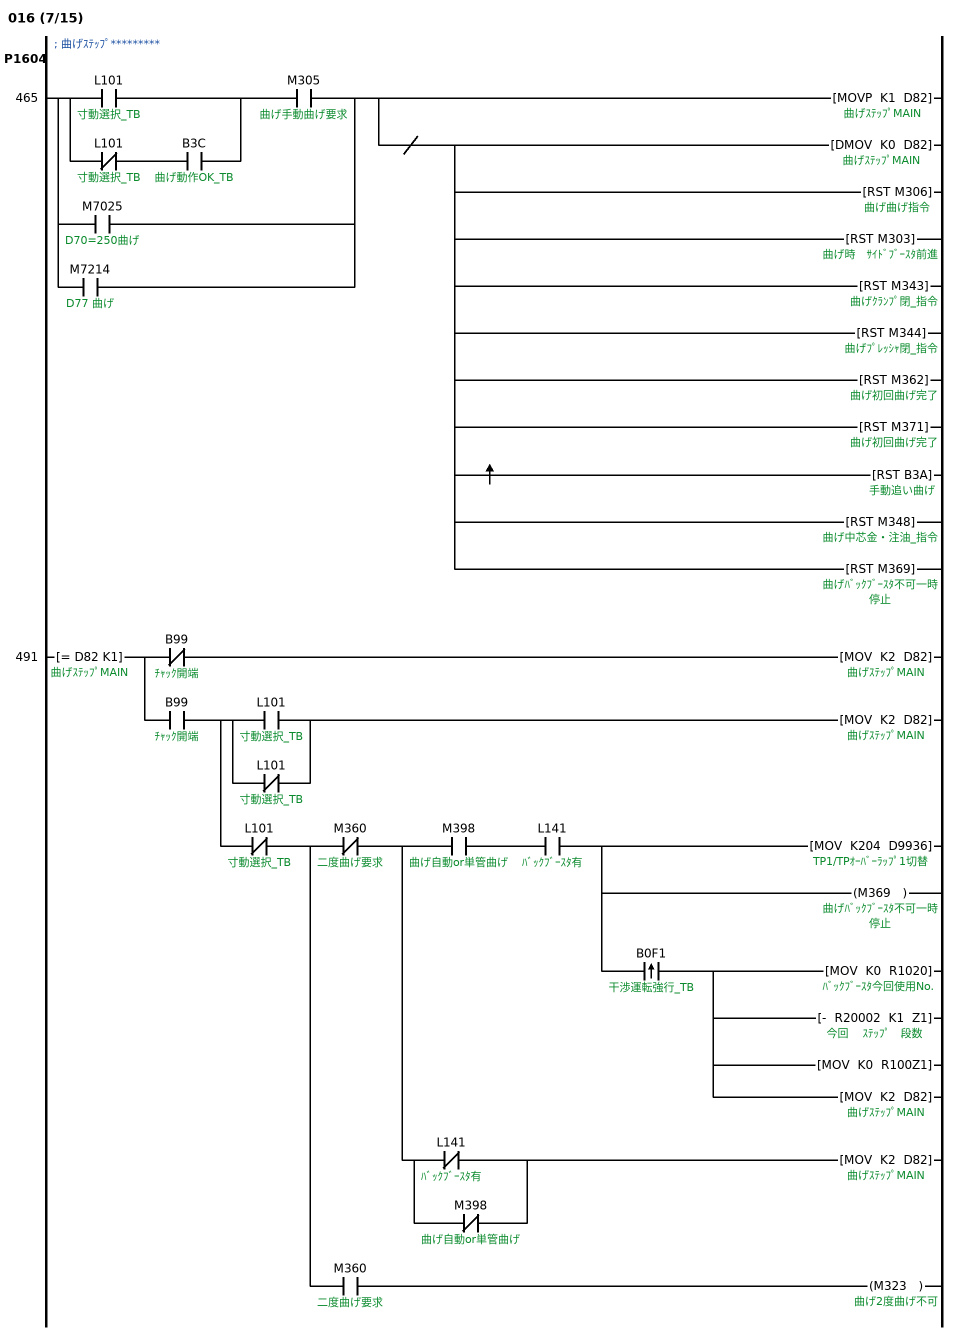
465   LD      L101  ; 寸動選択_TB
      LDI     L101  ; 寸動選択_TB
      AND     B3C  ; 曲げ動作OK_TB
      ORB
      AND     M305  ; 曲げ手動曲げ要求
      OR      M7025  ; D70=250曲げ
      OR      M7214  ; D77 曲げ
      MOVP    K1 D82  ; 曲げｽﾃｯﾌﾟMAIN
      INV
      DMOV    K0 D82
      RST     M306  ; 曲げ曲げ指令
      RST     M303  ; 曲げ時　ｻｲﾄﾞﾌﾞｰｽﾀ前進
      RST     M343  ; 曲げｸﾗﾝﾌﾟ閉_指令
      RST     M344  ; 曲げﾌﾟﾚｯｼｬ閉_指令
      RST     M362  ; 曲げ初回曲げ完了
      RST     M371  ; 曲げ初回曲げ完了
      MPS
      MEP
      RST     B3A  ; 手動追い曲げ
      MPP
      RST     M348  ; 曲げ中芯金・注油_指令
      RST     M369  ; 曲げﾊﾞｯｸﾌﾞｰｽﾀ不可一時停止
491   LD=     D82 K1  ; 曲げｽﾃｯﾌﾟMAIN
      MPS
      ANI     B99  ; ﾁｬｯｸ開端
      MOV     K2 D82
      MPP
      AND     B99  ; ﾁｬｯｸ開端
      MPS
      LD      L101  ; 寸動選択_TB
      ORI     L101  ; 寸動選択_TB
      ANB
      MOV     K2 D82
      MPP
      ANI     L101  ; 寸動選択_TB
      MPS
      ANI     M360  ; 二度曲げ要求
      MPS
      AND     M398  ; 曲げ自動or単管曲げ
      AND     L141  ; ﾊﾞｯｸﾌﾞｰｽﾀ有
      MOV     K204 D9936
      OUT     M369  ; 曲げﾊﾞｯｸﾌﾞｰｽﾀ不可一時停止
      ANDP    B0F1  ; 干渉運転強行_TB
      MOV     K0 R1020  ; ﾊﾞｯｸﾌﾞｰｽﾀ今回使用No.
      -       R20002 K1 Z1  ; 今回    ｽﾃｯﾌﾟ   段数
      MOV     K0 R100Z1
      MOV     K2 D82
      MPP
      LDI     L141  ; ﾊﾞｯｸﾌﾞｰｽﾀ有
      ORI     M398  ; 曲げ自動or単管曲げ
      ANB
      MOV     K2 D82
      MPP
      AND     M360  ; 二度曲げ要求
      OUT     M323  ; 曲げ2度曲げ不可
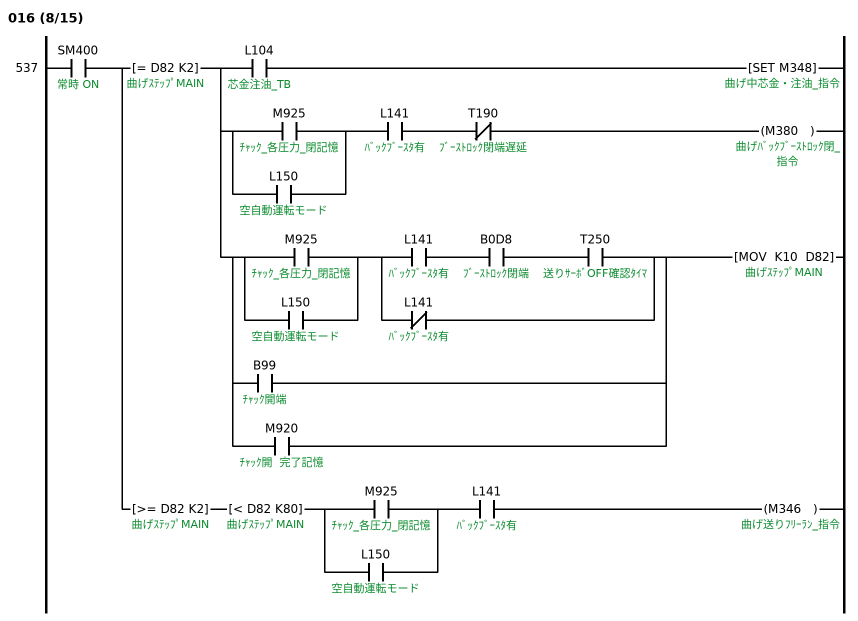
537   LD      SM400  ; 常時 ON
      MPS
      AND=    D82 K2  ; 曲げｽﾃｯﾌﾟMAIN
      MPS
      AND     L104  ; 芯金注油_TB
      SET     M348  ; 曲げ中芯金・注油_指令
      MRD
      LD      M925  ; ﾁｬｯｸ_各圧力_閉記憶
      OR      L150  ; 空自動運転モード
      ANB
      AND     L141  ; ﾊﾞｯｸﾌﾞｰｽﾀ有
      ANI     T190  ; ﾌﾞｰｽﾄﾛｯｸ閉端遅延
      OUT     M380  ; 曲げﾊﾞｯｸﾌﾞｰｽﾄﾛｯｸ閉_指令
      MPP
      LD      M925  ; ﾁｬｯｸ_各圧力_閉記憶
      OR      L150  ; 空自動運転モード
      LD      L141  ; ﾊﾞｯｸﾌﾞｰｽﾀ有
      AND     B0D8  ; ﾌﾞｰｽﾄﾛｯｸ閉端
      AND     T250  ; 送りｻｰﾎﾞOFF確認ﾀｲﾏ
      ORI     L141  ; ﾊﾞｯｸﾌﾞｰｽﾀ有
      ANB
      OR      B99  ; ﾁｬｯｸ開端
      OR      M920  ; ﾁｬｯｸ開  完了記憶
      ANB
      MOV     K10 D82
      MPP
      AND>=   D82 K2  ; 曲げｽﾃｯﾌﾟMAIN
      AND<    D82 K80  ; 曲げｽﾃｯﾌﾟMAIN
      LD      M925  ; ﾁｬｯｸ_各圧力_閉記憶
      OR      L150  ; 空自動運転モード
      ANB
      AND     L141  ; ﾊﾞｯｸﾌﾞｰｽﾀ有
      OUT     M346  ; 曲げ送りﾌﾘｰﾗﾝ_指令
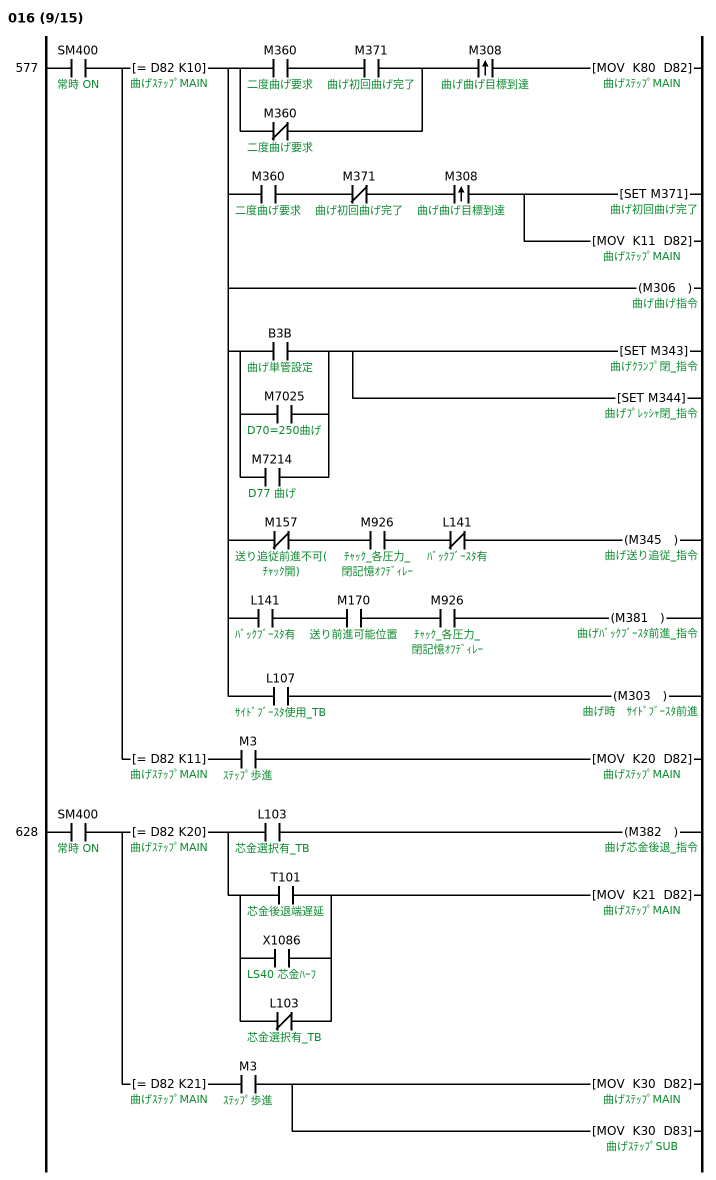
577   LD      SM400  ; 常時 ON
      MPS
      AND=    D82 K10  ; 曲げｽﾃｯﾌﾟMAIN
      MPS
      LD      M360  ; 二度曲げ要求
      AND     M371  ; 曲げ初回曲げ完了
      ORI     M360  ; 二度曲げ要求
      ANB
      ANDP    M308  ; 曲げ曲げ目標到達
      MOV     K80 D82
      MRD
      AND     M360  ; 二度曲げ要求
      ANI     M371  ; 曲げ初回曲げ完了
      ANDP    M308  ; 曲げ曲げ目標到達
      SET     M371  ; 曲げ初回曲げ完了
      MOV     K11 D82
      MPP
      OUT     M306  ; 曲げ曲げ指令
      MPS
      LD      B3B  ; 曲げ単管設定
      OR      M7025  ; D70=250曲げ
      OR      M7214  ; D77 曲げ
      ANB
      SET     M343  ; 曲げｸﾗﾝﾌﾟ閉_指令
      SET     M344  ; 曲げﾌﾟﾚｯｼｬ閉_指令
      MRD
      ANI     M157  ; 送り追従前進不可(ﾁｬｯｸ開)
      AND     M926  ; ﾁｬｯｸ_各圧力_閉記憶ｵﾌﾃﾞｨﾚｰ
      ANI     L141  ; ﾊﾞｯｸﾌﾞｰｽﾀ有
      OUT     M345  ; 曲げ送り追従_指令
      MRD
      AND     L141  ; ﾊﾞｯｸﾌﾞｰｽﾀ有
      AND     M170  ; 送り前進可能位置
      AND     M926  ; ﾁｬｯｸ_各圧力_閉記憶ｵﾌﾃﾞｨﾚｰ
      OUT     M381  ; 曲げﾊﾞｯｸﾌﾞｰｽﾀ前進_指令
      MPP
      AND     L107  ; ｻｲﾄﾞﾌﾞｰｽﾀ使用_TB
      OUT     M303  ; 曲げ時　ｻｲﾄﾞﾌﾞｰｽﾀ前進
      MPP
      AND=    D82 K11  ; 曲げｽﾃｯﾌﾟMAIN
      AND     M3  ; ｽﾃｯﾌﾟ歩進
      MOV     K20 D82
628   LD      SM400  ; 常時 ON
      MPS
      AND=    D82 K20  ; 曲げｽﾃｯﾌﾟMAIN
      MPS
      AND     L103  ; 芯金選択有_TB
      OUT     M382  ; 曲げ芯金後退_指令
      MPP
      LD      T101  ; 芯金後退端遅延
      OR      X1086  ; LS40 芯金ﾊｰﾌ
      ORI     L103  ; 芯金選択有_TB
      ANB
      MOV     K21 D82
      MPP
      AND=    D82 K21  ; 曲げｽﾃｯﾌﾟMAIN
      AND     M3  ; ｽﾃｯﾌﾟ歩進
      MOV     K30 D82
      MOV     K30 D83  ; 曲げｽﾃｯﾌﾟSUB
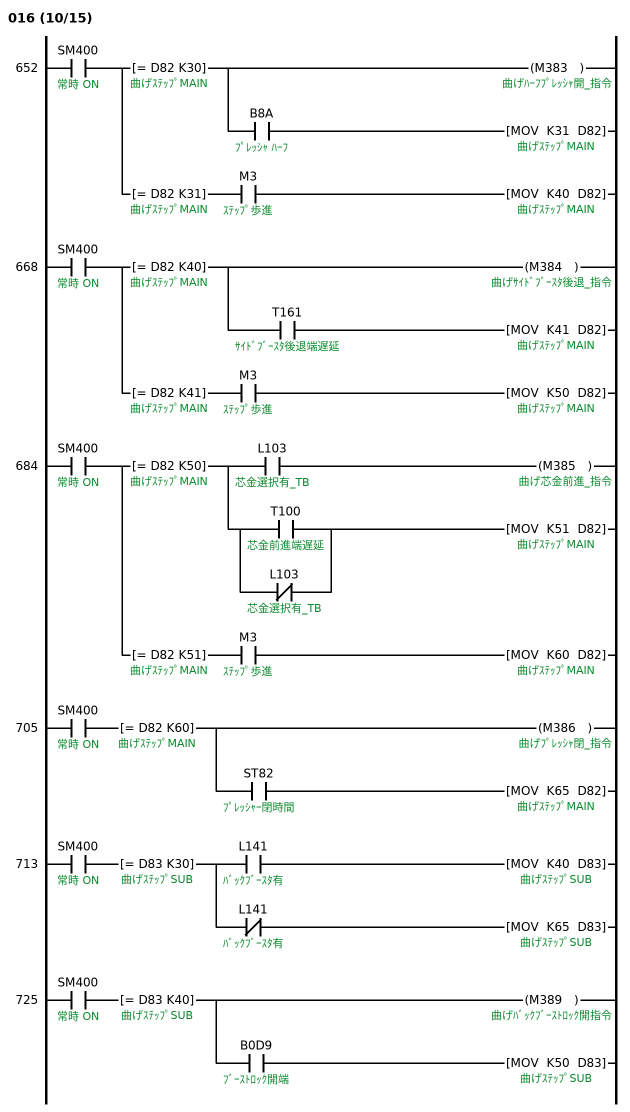
652   LD      SM400  ; 常時 ON
      MPS
      AND=    D82 K30  ; 曲げｽﾃｯﾌﾟMAIN
      OUT     M383  ; 曲げﾊｰﾌﾌﾟﾚｯｼｬ開_指令
      AND     B8A  ; ﾌﾟﾚｯｼｬ ﾊｰﾌ
      MOV     K31 D82
      MPP
      AND=    D82 K31  ; 曲げｽﾃｯﾌﾟMAIN
      AND     M3  ; ｽﾃｯﾌﾟ歩進
      MOV     K40 D82
668   LD      SM400  ; 常時 ON
      MPS
      AND=    D82 K40  ; 曲げｽﾃｯﾌﾟMAIN
      OUT     M384  ; 曲げｻｲﾄﾞﾌﾞｰｽﾀ後退_指令
      AND     T161  ; ｻｲﾄﾞﾌﾞｰｽﾀ後退端遅延
      MOV     K41 D82
      MPP
      AND=    D82 K41  ; 曲げｽﾃｯﾌﾟMAIN
      AND     M3  ; ｽﾃｯﾌﾟ歩進
      MOV     K50 D82
684   LD      SM400  ; 常時 ON
      MPS
      AND=    D82 K50  ; 曲げｽﾃｯﾌﾟMAIN
      MPS
      AND     L103  ; 芯金選択有_TB
      OUT     M385  ; 曲げ芯金前進_指令
      MPP
      LD      T100  ; 芯金前進端遅延
      ORI     L103  ; 芯金選択有_TB
      ANB
      MOV     K51 D82
      MPP
      AND=    D82 K51  ; 曲げｽﾃｯﾌﾟMAIN
      AND     M3  ; ｽﾃｯﾌﾟ歩進
      MOV     K60 D82
705   LD      SM400  ; 常時 ON
      AND=    D82 K60  ; 曲げｽﾃｯﾌﾟMAIN
      OUT     M386  ; 曲げﾌﾟﾚｯｼｬ閉_指令
      AND     ST82  ; ﾌﾟﾚｯｼｬｰ閉時間
      MOV     K65 D82
713   LD      SM400  ; 常時 ON
      AND=    D83 K30  ; 曲げｽﾃｯﾌﾟSUB
      MPS
      AND     L141  ; ﾊﾞｯｸﾌﾞｰｽﾀ有
      MOV     K40 D83
      MPP
      ANI     L141  ; ﾊﾞｯｸﾌﾞｰｽﾀ有
      MOV     K65 D83
725   LD      SM400  ; 常時 ON
      AND=    D83 K40  ; 曲げｽﾃｯﾌﾟSUB
      OUT     M389  ; 曲げﾊﾞｯｸﾌﾞｰｽﾄﾛｯｸ開指令
      AND     B0D9  ; ﾌﾞｰｽﾄﾛｯｸ開端
      MOV     K50 D83
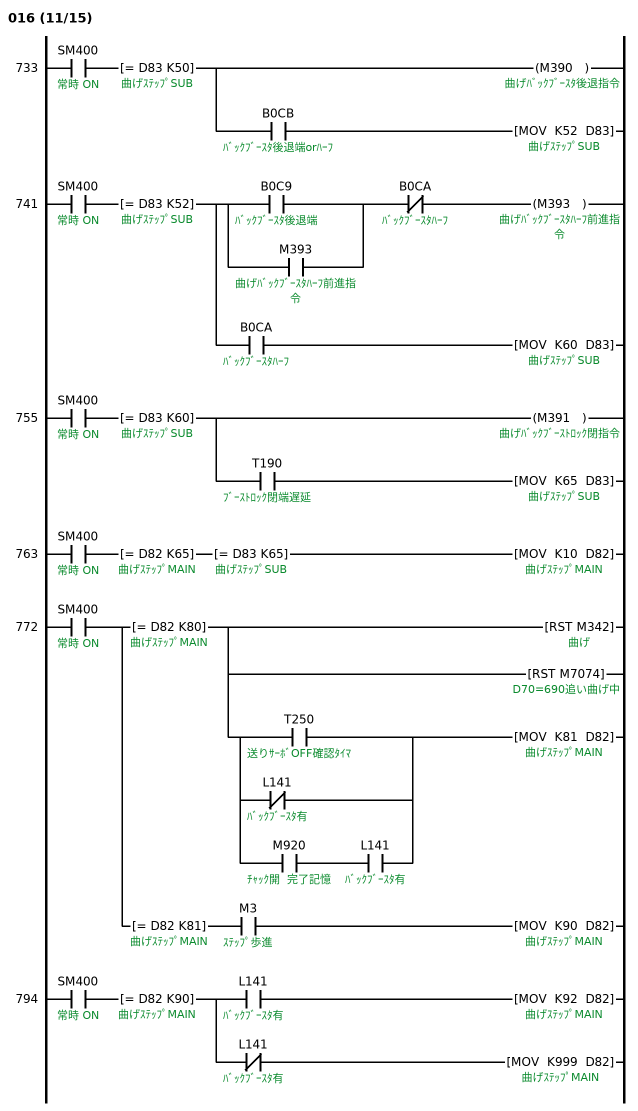
733   LD      SM400  ; 常時 ON
      AND=    D83 K50  ; 曲げｽﾃｯﾌﾟSUB
      OUT     M390  ; 曲げﾊﾞｯｸﾌﾞｰｽﾀ後退指令
      AND     B0CB  ; ﾊﾞｯｸﾌﾞｰｽﾀ後退端orﾊｰﾌ
      MOV     K52 D83
741   LD      SM400  ; 常時 ON
      AND=    D83 K52  ; 曲げｽﾃｯﾌﾟSUB
      MPS
      LD      B0C9  ; ﾊﾞｯｸﾌﾞｰｽﾀ後退端
      OR      M393  ; 曲げﾊﾞｯｸﾌﾞｰｽﾀﾊｰﾌ前進指令
      ANB
      ANI     B0CA  ; ﾊﾞｯｸﾌﾞｰｽﾀﾊｰﾌ
      OUT     M393  ; 曲げﾊﾞｯｸﾌﾞｰｽﾀﾊｰﾌ前進指令
      MPP
      AND     B0CA  ; ﾊﾞｯｸﾌﾞｰｽﾀﾊｰﾌ
      MOV     K60 D83
755   LD      SM400  ; 常時 ON
      AND=    D83 K60  ; 曲げｽﾃｯﾌﾟSUB
      OUT     M391  ; 曲げﾊﾞｯｸﾌﾞｰｽﾄﾛｯｸ閉指令
      AND     T190  ; ﾌﾞｰｽﾄﾛｯｸ閉端遅延
      MOV     K65 D83
763   LD      SM400  ; 常時 ON
      AND=    D82 K65  ; 曲げｽﾃｯﾌﾟMAIN
      AND=    D83 K65  ; 曲げｽﾃｯﾌﾟSUB
      MOV     K10 D82
772   LD      SM400  ; 常時 ON
      MPS
      AND=    D82 K80  ; 曲げｽﾃｯﾌﾟMAIN
      RST     M342  ; 曲げ
      RST     M7074  ; D70=690追い曲げ中
      LD      T250  ; 送りｻｰﾎﾞOFF確認ﾀｲﾏ
      ORI     L141  ; ﾊﾞｯｸﾌﾞｰｽﾀ有
      LD      M920  ; ﾁｬｯｸ開  完了記憶
      AND     L141  ; ﾊﾞｯｸﾌﾞｰｽﾀ有
      ORB
      ANB
      MOV     K81 D82
      MPP
      AND=    D82 K81  ; 曲げｽﾃｯﾌﾟMAIN
      AND     M3  ; ｽﾃｯﾌﾟ歩進
      MOV     K90 D82
794   LD      SM400  ; 常時 ON
      AND=    D82 K90  ; 曲げｽﾃｯﾌﾟMAIN
      MPS
      AND     L141  ; ﾊﾞｯｸﾌﾞｰｽﾀ有
      MOV     K92 D82
      MPP
      ANI     L141  ; ﾊﾞｯｸﾌﾞｰｽﾀ有
      MOV     K999 D82
